LIN {X 0,Y 270.162,Z 852.684,A -85,B 0,C 180,E1 7695.271,E2 7695.271} C_VEL
LIN {X 0,Y 259.155,Z 871.54,A -85,B 0,C 180,E1 7693.362,E2 7693.362} C_VEL
LIN {X 0,Y 247.271,Z 889.429,A -85,B 0,C 180,E1 7691.066,E2 7691.066} C_VEL
LIN {X 0,Y 235.05,Z 906.14,A -85,B 0,C 180,E1 7688.382,E2 7688.382} C_VEL
LIN {X 0,Y 222.958,Z 921.018,A -85,B 0,C 180,E1 7685.334,E2 7685.334} C_VEL
LIN {X 0,Y 210.174,Z 935.544,A -85,B 0,C 180,E1 7681.543,E2 7681.543} C_VEL
LIN {X 0,Y 198.279,Z 948.046,A -85,B 0,C 180,E1 7677.304,E2 7677.304} C_VEL
LIN {X 0,Y 186.376,Z 959.885,A -85,B 0,C 180,E1 7672.046,E2 7672.046} C_VEL
LIN {X 0,Y 176.439,Z 969.458,A -85,B 0,C 180,E1 7666.449,E2 7666.449} C_VEL
LIN {X 0,Y 167.3,Z 978.146,A -85,B 0,C 180,E1 7659.622,E2 7659.622} C_VEL
LIN {X 0,Y 160.302,Z 985.227,A -85,B 0,C 180,E1 7652.134,E2 7652.134} C_VEL
LIN {X 0,Y 155.686,Z 990.327,A -85,B 0,C 180,E1 7644.461,E2 7644.461} C_VEL
LIN {X 0,Y 153.174,Z 993.985,A -85,B 0,C 180,E1 7636.782,E2 7636.782} C_VEL
LIN {X 0,Y 152.199,Z 996.255,A -85,B 0,C 180,E1 7628.889,E2 7628.889} C_VEL
LIN {X 0,Y 152.061,Z 997.122,A -85,B 0,C 180,E1 7623.007,E2 7623.007} C_VEL
LIN {X 0,Y 152.146,Z 997.282,A -85,B 0,C 180,E1 7616.932,E2 7616.932} C_VEL
LIN {X 0,Y 152.676,Z 996.667,A -85,B 0,C 180,E1 7610.549,E2 7610.549} C_VEL
LIN {X 0,Y 154.828,Z 994.686,A -85,B 0,C 180,E1 7602.194,E2 7602.194} C_VEL
LIN {X 0,Y 159.181,Z 991.12,A -85,B 0,C 180,E1 7593.974,E2 7593.974} C_VEL
LIN {X 0,Y 166.545,Z 985.817,A -85,B 0,C 180,E1 7585.753,E2 7585.753} C_VEL
LIN {X 0,Y 176.186,Z 979.026,A -85,B 0,C 180,E1 7578.531,E2 7578.531} C_VEL
LIN {X 0,Y 188.917,Z 969.957,A -85,B 0,C 180,E1 7571.693,E2 7571.693} C_VEL
LIN {X 0,Y 203.113,Z 959.499,A -85,B 0,C 180,E1 7566.019,E2 7566.019} C_VEL
LIN {X 0,Y 218.195,Z 947.498,A -85,B 0,C 180,E1 7561.314,E2 7561.314} C_VEL
LIN {X 0,Y 234.781,Z 933.271,A -85,B 0,C 180,E1 7557.194,E2 7557.194} C_VEL
LIN {X 0,Y 250.793,Z 918.312,A -85,B 0,C 180,E1 7553.948,E2 7553.948} C_VEL
LIN {X 0,Y 266.015,Z 902.433,A -85,B 0,C 180,E1 7551.34,E2 7551.34} C_VEL
LIN {X 0,Y 281.745,Z 884.288,A -85,B 0,C 180,E1 7549.046,E2 7549.046} C_VEL
LIN {X 0,Y 295.555,Z 866.409,A -85,B 0,C 180,E1 7547.298,E2 7547.298} C_VEL
LIN {X 0,Y 302.047,Z 857.131,A -85,B 0,C 180,E1 7546.521,E2 7546.521} C_VEL
LIN {X 0,Y 290.09,Z 874.11,A -85,B 0,C 180,E1 7545.216,E2 7545.216} C_VEL
LIN {X 0,Y 285.508,Z 880.165,A -85,B 0,C 180,E1 7544.883,E2 7544.883} C_VEL
LIN {X 0,Y 272.533,Z 895.474,A -85,B 0,C 180,E1 7544.622,E2 7544.622} C_VEL
LIN {X 0,Y 267.468,Z 900.978,A -85,B 0,C 180,E1 7544.201,E2 7544.201} C_VEL
LIN {X 0,Y 252.345,Z 916.917,A -85,B 0,C 180,E1 7541.995,E2 7541.995} C_VEL
LIN {X 0,Y 235.551,Z 933.117,A -85,B 0,C 180,E1 7539.058,E2 7539.058} C_VEL
LIN {X 0,Y 220.329,Z 946.567,A -85,B 0,C 180,E1 7535.817,E2 7535.817} C_VEL
LIN {X 0,Y 203.797,Z 960.142,A -85,B 0,C 180,E1 7531.44,E2 7531.44} C_VEL
LIN {X 0,Y 189.339,Z 971.334,A -85,B 0,C 180,E1 7526.563,E2 7526.563} C_VEL
LIN {X 0,Y 175.331,Z 981.675,A -85,B 0,C 180,E1 7520.354,E2 7520.354} C_VEL
LIN {X 0,Y 163.608,Z 990.335,A -85,B 0,C 180,E1 7513.206,E2 7513.206} C_VEL
LIN {X 0,Y 154.524,Z 997.124,A -85,B 0,C 180,E1 7505.173,E2 7505.173} C_VEL
LIN {X 0,Y 148.144,Z 1002.572,A -85,B 0,C 180,E1 7496.033,E2 7496.033} C_VEL
LIN {X 0,Y 145.093,Z 1005.814,A -85,B 0,C 180,E1 7487.662,E2 7487.662} C_VEL
LIN {X 0,Y 144.092,Z 1007.682,A -85,B 0,C 180,E1 7479.831,E2 7479.831} C_VEL
LIN {X 0,Y 144.042,Z 1008.346,A -85,B 0,C 180,E1 7472.797,E2 7472.797} C_VEL
LIN {X 0,Y 144.047,Z 1008.068,A -85,B 0,C 180,E1 7466.829,E2 7466.829} C_VEL
LIN {X 0,Y 144.115,Z 1006.784,A -85,B 0,C 180,E1 7460.024,E2 7460.024} C_VEL
LIN {X 0,Y 145.002,Z 1004.362,A -85,B 0,C 180,E1 7452.765,E2 7452.765} C_VEL
LIN {X 0,Y 147.505,Z 1000.647,A -85,B 0,C 180,E1 7445.163,E2 7445.163} C_VEL
LIN {X 0,Y 152.755,Z 994.682,A -85,B 0,C 180,E1 7436.66,E2 7436.66} C_VEL
LIN {X 0,Y 159.808,Z 987.715,A -85,B 0,C 180,E1 7429.423,E2 7429.423} C_VEL
LIN {X 0,Y 169.417,Z 978.623,A -85,B 0,C 180,E1 7422.48,E2 7422.48} C_VEL
LIN {X 0,Y 180.465,Z 968.26,A -85,B 0,C 180,E1 7416.566,E2 7416.566} C_VEL
LIN {X 0,Y 192.416,Z 956.466,A -85,B 0,C 180,E1 7411.569,E2 7411.569} C_VEL
LIN {X 0,Y 205.608,Z 942.836,A -85,B 0,C 180,E1 7407.16,E2 7407.16} C_VEL
LIN {X 0,Y 218.285,Z 928.559,A -85,B 0,C 180,E1 7403.662,E2 7403.662} C_VEL
LIN {X 0,Y 231.669,Z 912.241,A -85,B 0,C 180,E1 7400.548,E2 7400.548} C_VEL
LIN {X 0,Y 243.409,Z 896.383,A -85,B 0,C 180,E1 7398.19,E2 7398.19} C_VEL
LIN {X 0,Y 256.695,Z 876.382,A -85,B 0,C 180,E1 7395.859,E2 7395.859} C_VEL
LIN {X 0,Y 268.011,Z 857.211,A -85,B 0,C 180,E1 7394.113,E2 7394.113} C_VEL
LIN {X 0,Y 278.538,Z 836.599,A -85,B 0,C 180,E1 7392.648,E2 7392.648} C_VEL
LIN {X 0,Y 288.142,Z 814.942,A -85,B 0,C 180,E1 7391.439,E2 7391.439} C_VEL
LIN {X 0,Y 295.909,Z 794.1,A -85,B 0,C 180,E1 7390.539,E2 7390.539} C_VEL
LIN {X 0,Y 303.26,Z 770.05,A -85,B 0,C 180,E1 7389.753,E2 7389.753} C_VEL
LIN {X 0,Y 308.805,Z 746.808,A -85,B 0,C 180,E1 7389.177,E2 7389.177} C_VEL
LIN {X 0,Y 312.638,Z 723.003,A -85,B 0,C 180,E1 7388.694,E2 7388.694} C_VEL
LIN {X 0,Y 326.224,Z 603.459,A -85,B 0,C 180,E1 7386.559,E2 7386.559} C_VEL
LIN {X 0,Y 322.526,Z 597.162,A -85,B 0,C 180,E1 7383.198,E2 7383.198} C_VEL
LIN {X 0,Y 320.23,Z 593.384,A -85,B 0,C 180,E1 7380.715,E2 7380.715} C_VEL
LIN {X 0,Y 317.941,Z 589.485,A -85,B 0,C 180,E1 7377.656,E2 7377.656} C_VEL
LIN {X 0,Y 315.609,Z 585.291,A -85,B 0,C 180,E1 7373.268,E2 7373.268} C_VEL
LIN {X 0,Y 313.967,Z 583.652,A -85,B 0,C 180,E1 7367.119,E2 7367.119} C_VEL
LIN {X 0,Y 314.171,Z 583.904,A -85,B 0,C 180,E1 7362.592,E2 7362.592} C_VEL
LIN {X 0,Y 315.683,Z 585.371,A -85,B 0,C 180,E1 7357.857,E2 7357.857} C_VEL
LIN {X 0,Y 318.646,Z 590.582,A -85,B 0,C 180,E1 7352.608,E2 7352.608} C_VEL
LIN {X 0,Y 321.436,Z 595.282,A -85,B 0,C 180,E1 7349.222,E2 7349.222} C_VEL
LIN {X 0,Y 324.307,Z 600.175,A -85,B 0,C 180,E1 7346.387,E2 7346.387} C_VEL
LIN {X 0,Y 325.927,Z 603.009,A -85,B 0,C 180,E1 7344.966,E2 7344.966} C_VEL
LIN {X 0,Y 312.184,Z 722.288,A -85,B 0,C 180,E1 7342.851,E2 7342.851} C_VEL
LIN {X 0,Y 307.763,Z 746.045,A -85,B 0,C 180,E1 7342.322,E2 7342.322} C_VEL
LIN {X 0,Y 302.328,Z 768.096,A -85,B 0,C 180,E1 7341.675,E2 7341.675} C_VEL
LIN {X 0,Y 295.325,Z 790.127,A -85,B 0,C 180,E1 7340.821,E2 7340.821} C_VEL
LIN {X 0,Y 286.506,Z 813.129,A -85,B 0,C 180,E1 7339.676,E2 7339.676} C_VEL
LIN {X 0,Y 277.365,Z 833.259,A -85,B 0,C 180,E1 7338.406,E2 7338.406} C_VEL
LIN {X 0,Y 266.708,Z 853.445,A -85,B 0,C 180,E1 7336.804,E2 7336.804} C_VEL
LIN {X 0,Y 255.463,Z 872.302,A -85,B 0,C 180,E1 7334.936,E2 7334.936} C_VEL
LIN {X 0,Y 243.293,Z 890.156,A -85,B 0,C 180,E1 7332.683,E2 7332.683} C_VEL
LIN {X 0,Y 230.369,Z 907.254,A -85,B 0,C 180,E1 7329.956,E2 7329.956} C_VEL
LIN {X 0,Y 217.938,Z 922.067,A -85,B 0,C 180,E1 7326.93,E2 7326.93} C_VEL
LIN {X 0,Y 204.075,Z 937.188,A -85,B 0,C 180,E1 7322.934,E2 7322.934} C_VEL
LIN {X 0,Y 191.817,Z 949.595,A -85,B 0,C 180,E1 7318.645,E2 7318.645} C_VEL
LIN {X 0,Y 179.49,Z 961.211,A -85,B 0,C 180,E1 7313.286,E2 7313.286} C_VEL
LIN {X 0,Y 168.711,Z 971.103,A -85,B 0,C 180,E1 7307.225,E2 7307.225} C_VEL
LIN {X 0,Y 159.593,Z 979.245,A -85,B 0,C 180,E1 7300.379,E2 7300.379} C_VEL
LIN {X 0,Y 152.097,Z 986.35,A -85,B 0,C 180,E1 7292.224,E2 7292.224} C_VEL
LIN {X 0,Y 147.629,Z 991.075,A -85,B 0,C 180,E1 7284.547,E2 7284.547} C_VEL
LIN {X 0,Y 145.011,Z 994.73,A -85,B 0,C 180,E1 7276.023,E2 7276.023} C_VEL
LIN {X 0,Y 144.201,Z 996.581,A -85,B 0,C 180,E1 7268.853,E2 7268.853} C_VEL
LIN {X 0,Y 144.069,Z 997.435,A -85,B 0,C 180,E1 7262.669,E2 7262.669} C_VEL
LIN {X 0,Y 144.157,Z 997.607,A -85,B 0,C 180,E1 7256.762,E2 7256.762} C_VEL
LIN {X 0,Y 144.755,Z 997.043,A -85,B 0,C 180,E1 7250.017,E2 7250.017} C_VEL
LIN {X 0,Y 147.012,Z 995.246,A -85,B 0,C 180,E1 7241.556,E2 7241.556} C_VEL
LIN {X 0,Y 151.941,Z 991.659,A -85,B 0,C 180,E1 7232.597,E2 7232.597} C_VEL
LIN {X 0,Y 159.924,Z 986.487,A -85,B 0,C 180,E1 7224.083,E2 7224.083} C_VEL
LIN {X 0,Y 170.496,Z 979.611,A -85,B 0,C 180,E1 7216.529,E2 7216.529} C_VEL
LIN {X 0,Y 184.493,Z 970.332,A -85,B 0,C 180,E1 7209.435,E2 7209.435} C_VEL
LIN {X 0,Y 199.438,Z 959.955,A -85,B 0,C 180,E1 7203.823,E2 7203.823} C_VEL
LIN {X 0,Y 215.272,Z 947.978,A -85,B 0,C 180,E1 7199.203,E2 7199.203} C_VEL
LIN {X 0,Y 232.015,Z 934.265,A -85,B 0,C 180,E1 7195.304,E2 7195.304} C_VEL
LIN {X 0,Y 248.645,Z 919.344,A -85,B 0,C 180,E1 7192.143,E2 7192.143} C_VEL
LIN {X 0,Y 264.823,Z 903.077,A -85,B 0,C 180,E1 7189.56,E2 7189.56} C_VEL
LIN {X 0,Y 280.736,Z 885.326,A -85,B 0,C 180,E1 7187.405,E2 7187.405} C_VEL
LIN {X 0,Y 287.244,Z 877.461,A -85,B 0,C 180,E1 7186.594,E2 7186.594} C_VEL
LIN {X 0,Y 273.077,Z 894.577,A -85,B 0,C 180,E1 7184.933,E2 7184.933} C_VEL
LIN {X 0,Y 267.468,Z 900.978,A -85,B 0,C 180,E1 7184.201,E2 7184.201} C_VEL
LIN {X 0,Y 262.279,Z 906.461,A -85,B 0,C 180,E1 7183.741,E2 7183.741} C_VEL
LIN {X 0,Y 247.934,Z 920.355,A -85,B 0,C 180,E1 7183.165,E2 7183.165} C_VEL
LIN {X 0,Y 242.565,Z 925.2,A -85,B 0,C 180,E1 7182.583,E2 7182.583} C_VEL
LIN {X 0,Y 225.228,Z 940.622,A -85,B 0,C 180,E1 7179.471,E2 7179.471} C_VEL
LIN {X 0,Y 208.402,Z 954.183,A -85,B 0,C 180,E1 7175.739,E2 7175.739} C_VEL
LIN {X 0,Y 190.481,Z 967.605,A -85,B 0,C 180,E1 7170.631,E2 7170.631} C_VEL
LIN {X 0,Y 174.945,Z 978.613,A -85,B 0,C 180,E1 7164.745,E2 7164.745} C_VEL
LIN {X 0,Y 161.697,Z 987.525,A -85,B 0,C 180,E1 7157.918,E2 7157.918} C_VEL
LIN {X 0,Y 150.354,Z 995.281,A -85,B 0,C 180,E1 7149.522,E2 7149.522} C_VEL
LIN {X 0,Y 142.712,Z 1000.798,A -85,B 0,C 180,E1 7140.773,E2 7140.773} C_VEL
LIN {X 0,Y 137.876,Z 1004.997,A -85,B 0,C 180,E1 7130.697,E2 7130.697} C_VEL
LIN {X 0,Y 136.278,Z 1007.009,A -85,B 0,C 180,E1 7122.636,E2 7122.636} C_VEL
LIN {X 0,Y 136.032,Z 1007.885,A -85,B 0,C 180,E1 7115.496,E2 7115.496} C_VEL
LIN {X 0,Y 136.079,Z 1007.881,A -85,B 0,C 180,E1 7109.171,E2 7109.171} C_VEL
LIN {X 0,Y 136.04,Z 1007.111,A -85,B 0,C 180,E1 7102.833,E2 7102.833} C_VEL
LIN {X 0,Y 136.628,Z 1005.093,A -85,B 0,C 180,E1 7094.739,E2 7094.739} C_VEL
LIN {X 0,Y 139.031,Z 1001.332,A -85,B 0,C 180,E1 7085.966,E2 7085.966} C_VEL
LIN {X 0,Y 143.696,Z 996.28,A -85,B 0,C 180,E1 7077.619,E2 7077.619} C_VEL
LIN {X 0,Y 150.992,Z 989.347,A -85,B 0,C 180,E1 7069.555,E2 7069.555} C_VEL
LIN {X 0,Y 160.748,Z 980.735,A -85,B 0,C 180,E1 7062.201,E2 7062.201} C_VEL
LIN {X 0,Y 172.157,Z 970.459,A -85,B 0,C 180,E1 7055.914,E2 7055.914} C_VEL
LIN {X 0,Y 185.372,Z 958.223,A -85,B 0,C 180,E1 7050.367,E2 7050.367} C_VEL
LIN {X 0,Y 198.608,Z 945.144,A -85,B 0,C 180,E1 7045.974,E2 7045.974} C_VEL
LIN {X 0,Y 212.657,Z 930.054,A -85,B 0,C 180,E1 7042.171,E2 7042.171} C_VEL
LIN {X 0,Y 226.361,Z 914.035,A -85,B 0,C 180,E1 7039.076,E2 7039.076} C_VEL
LIN {X 0,Y 239.354,Z 896.996,A -85,B 0,C 180,E1 7036.559,E2 7036.559} C_VEL
LIN {X 0,Y 252.328,Z 878.125,A -85,B 0,C 180,E1 7034.377,E2 7034.377} C_VEL
LIN {X 0,Y 263.801,Z 859.218,A -85,B 0,C 180,E1 7032.674,E2 7032.674} C_VEL
LIN {X 0,Y 274.861,Z 838.315,A -85,B 0,C 180,E1 7031.2,E2 7031.2} C_VEL
LIN {X 0,Y 284.294,Z 817.819,A -85,B 0,C 180,E1 7030.065,E2 7030.065} C_VEL
LIN {X 0,Y 292.631,Z 796.13,A -85,B 0,C 180,E1 7029.138,E2 7029.138} C_VEL
LIN {X 0,Y 299.852,Z 773.653,A -85,B 0,C 180,E1 7028.402,E2 7028.402} C_VEL
LIN {X 0,Y 305.465,Z 751.2,A -85,B 0,C 180,E1 7027.85,E2 7027.85} C_VEL
LIN {X 0,Y 309.952,Z 726.087,A -85,B 0,C 180,E1 7027.337,E2 7027.337} C_VEL
LIN {X 0,Y 323.595,Z 609.157,A -85,B 0,C 180,E1 7025.274,E2 7025.274} C_VEL
LIN {X 0,Y 320.64,Z 604.095,A -85,B 0,C 180,E1 7022.412,E2 7022.412} C_VEL
LIN {X 0,Y 318.812,Z 601.022,A -85,B 0,C 180,E1 7020.359,E2 7020.359} C_VEL
LIN {X 0,Y 316.708,Z 597.319,A -85,B 0,C 180,E1 7017.466,E2 7017.466} C_VEL
LIN {X 0,Y 314.42,Z 593.131,A -85,B 0,C 180,E1 7013.059,E2 7013.059} C_VEL
LIN {X 0,Y 312.859,Z 591.556,A -85,B 0,C 180,E1 7006.884,E2 7006.884} C_VEL
LIN {X 0,Y 313.119,Z 591.891,A -85,B 0,C 180,E1 7002.34,E2 7002.34} C_VEL
LIN {X 0,Y 314.525,Z 593.322,A -85,B 0,C 180,E1 6997.968,E2 6997.968} C_VEL
LIN {X 0,Y 317.37,Z 598.423,A -85,B 0,C 180,E1 6992.817,E2 6992.817} C_VEL
LIN {X 0,Y 320.048,Z 603.022,A -85,B 0,C 180,E1 6989.501,E2 6989.501} C_VEL
LIN {X 0,Y 322.87,Z 607.937,A -85,B 0,C 180,E1 6986.654,E2 6986.654} C_VEL
LIN {X 0,Y 323.29,Z 608.915,A -85,B 0,C 180,E1 6986.237,E2 6986.237} C_VEL
LIN {X 0,Y 309.904,Z 722.563,A -85,B 0,C 180,E1 6984.262,E2 6984.262} C_VEL
LIN {X 0,Y 305.413,Z 746.343,A -85,B 0,C 180,E1 6983.751,E2 6983.751} C_VEL
LIN {X 0,Y 299.702,Z 769.038,A -85,B 0,C 180,E1 6983.103,E2 6983.103} C_VEL
LIN {X 0,Y 293.013,Z 789.796,A -85,B 0,C 180,E1 6982.328,E2 6982.328} C_VEL
LIN {X 0,Y 284.468,Z 811.998,A -85,B 0,C 180,E1 6981.275,E2 6981.275} C_VEL
LIN {X 0,Y 275.151,Z 832.32,A -85,B 0,C 180,E1 6980.05,E2 6980.05} C_VEL
LIN {X 0,Y 263.86,Z 853.451,A -85,B 0,C 180,E1 6978.439,E2 6978.439} C_VEL
LIN {X 0,Y 251.96,Z 872.97,A -85,B 0,C 180,E1 6976.557,E2 6976.557} C_VEL
LIN {X 0,Y 239.505,Z 890.788,A -85,B 0,C 180,E1 6974.355,E2 6974.355} C_VEL
LIN {X 0,Y 225.865,Z 908.325,A -85,B 0,C 180,E1 6971.595,E2 6971.595} C_VEL
LIN {X 0,Y 213.094,Z 923.108,A -85,B 0,C 180,E1 6968.6,E2 6968.6} C_VEL
LIN {X 0,Y 199.488,Z 937.426,A -85,B 0,C 180,E1 6964.834,E2 6964.834} C_VEL
LIN {X 0,Y 186.739,Z 949.846,A -85,B 0,C 180,E1 6960.562,E2 6960.562} C_VEL
LIN {X 0,Y 173.848,Z 961.488,A -85,B 0,C 180,E1 6955.176,E2 6955.176} C_VEL
LIN {X 0,Y 162.484,Z 971.404,A -85,B 0,C 180,E1 6949.023,E2 6949.023} C_VEL
LIN {X 0,Y 152.887,Z 979.481,A -85,B 0,C 180,E1 6942.068,E2 6942.068} C_VEL
LIN {X 0,Y 145.085,Z 986.383,A -85,B 0,C 180,E1 6933.94,E2 6933.94} C_VEL
LIN {X 0,Y 140.126,Z 991.169,A -85,B 0,C 180,E1 6925.896,E2 6925.896} C_VEL
LIN {X 0,Y 137.17,Z 994.917,A -85,B 0,C 180,E1 6916.928,E2 6916.928} C_VEL
LIN {X 0,Y 136.202,Z 996.904,A -85,B 0,C 180,E1 6908.802,E2 6908.802} C_VEL
LIN {X 0,Y 136.075,Z 997.737,A -85,B 0,C 180,E1 6902.411,E2 6902.411} C_VEL
LIN {X 0,Y 136.189,Z 997.917,A -85,B 0,C 180,E1 6896.062,E2 6896.062} C_VEL
LIN {X 0,Y 136.958,Z 997.335,A -85,B 0,C 180,E1 6888.762,E2 6888.762} C_VEL
LIN {X 0,Y 139.749,Z 995.455,A -85,B 0,C 180,E1 6879.553,E2 6879.553} C_VEL
LIN {X 0,Y 145.197,Z 991.97,A -85,B 0,C 180,E1 6870.577,E2 6870.577} C_VEL
LIN {X 0,Y 154.127,Z 986.734,A -85,B 0,C 180,E1 6861.703,E2 6861.703} C_VEL
LIN {X 0,Y 165.137,Z 980.154,A -85,B 0,C 180,E1 6854.326,E2 6854.326} C_VEL
LIN {X 0,Y 179.687,Z 971.191,A -85,B 0,C 180,E1 6847.354,E2 6847.354} C_VEL
LIN {X 0,Y 194.432,Z 961.539,A -85,B 0,C 180,E1 6842.064,E2 6842.064} C_VEL
LIN {X 0,Y 210.567,Z 950.06,A -85,B 0,C 180,E1 6837.552,E2 6837.552} C_VEL
LIN {X 0,Y 227.311,Z 937.188,A -85,B 0,C 180,E1 6833.819,E2 6833.819} C_VEL
LIN {X 0,Y 243.785,Z 923.052,A -85,B 0,C 180,E1 6830.797,E2 6830.797} C_VEL
LIN {X 0,Y 260.438,Z 907.351,A -85,B 0,C 180,E1 6828.253,E2 6828.253} C_VEL
LIN {X 0,Y 272.321,Z 894.975,A -85,B 0,C 180,E1 6826.668,E2 6826.668} C_VEL
LIN {X 0,Y 255.283,Z 912.982,A -85,B 0,C 180,E1 6824.489,E2 6824.489} C_VEL
LIN {X 0,Y 242.565,Z 925.2,A -85,B 0,C 180,E1 6822.583,E2 6822.583} C_VEL
LIN {X 0,Y 237.076,Z 930.151,A -85,B 0,C 180,E1 6821.949,E2 6821.949} C_VEL
LIN {X 0,Y 221.601,Z 942.319,A -85,B 0,C 180,E1 6820.953,E2 6820.953} C_VEL
LIN {X 0,Y 215.982,Z 946.624,A -85,B 0,C 180,E1 6820.166,E2 6820.166} C_VEL
LIN {X 0,Y 198.015,Z 960.01,A -85,B 0,C 180,E1 6816.072,E2 6816.072} C_VEL
LIN {X 0,Y 180.739,Z 972.007,A -85,B 0,C 180,E1 6810.95,E2 6810.95} C_VEL
LIN {X 0,Y 165.19,Z 981.995,A -85,B 0,C 180,E1 6804.813,E2 6804.813} C_VEL
LIN {X 0,Y 150.825,Z 990.968,A -85,B 0,C 180,E1 6796.835,E2 6796.835} C_VEL
LIN {X 0,Y 140.443,Z 997.516,A -85,B 0,C 180,E1 6788.285,E2 6788.285} C_VEL
LIN {X 0,Y 132.973,Z 1002.569,A -85,B 0,C 180,E1 6778.289,E2 6778.289} C_VEL
LIN {X 0,Y 129.324,Z 1005.632,A -85,B 0,C 180,E1 6768.962,E2 6768.962} C_VEL
LIN {X 0,Y 128.086,Z 1007.33,A -85,B 0,C 180,E1 6759.448,E2 6759.448} C_VEL
LIN {X 0,Y 128.07,Z 1007.674,A -85,B 0,C 180,E1 6752.173,E2 6752.173} C_VEL
LIN {X 0,Y 128.056,Z 1007.296,A -85,B 0,C 180,E1 6745.984,E2 6745.984} C_VEL
LIN {X 0,Y 128.18,Z 1006.002,A -85,B 0,C 180,E1 6738.769,E2 6738.769} C_VEL
LIN {X 0,Y 129.433,Z 1003.5,A -85,B 0,C 180,E1 6730.614,E2 6730.614} C_VEL
LIN {X 0,Y 133.113,Z 999.24,A -85,B 0,C 180,E1 6721.283,E2 6721.283} C_VEL
LIN {X 0,Y 139.451,Z 993.223,A -85,B 0,C 180,E1 6712.468,E2 6712.468} C_VEL
LIN {X 0,Y 148.404,Z 985.668,A -85,B 0,C 180,E1 6704.444,E2 6704.444} C_VEL
LIN {X 0,Y 159.468,Z 976.363,A -85,B 0,C 180,E1 6697.457,E2 6697.457} C_VEL
LIN {X 0,Y 172.921,Z 964.773,A -85,B 0,C 180,E1 6691.179,E2 6691.179} C_VEL
LIN {X 0,Y 186.317,Z 952.571,A -85,B 0,C 180,E1 6686.363,E2 6686.363} C_VEL
LIN {X 0,Y 200.413,Z 938.594,A -85,B 0,C 180,E1 6682.281,E2 6682.281} C_VEL
LIN {X 0,Y 214.524,Z 923.448,A -85,B 0,C 180,E1 6678.921,E2 6678.921} C_VEL
LIN {X 0,Y 227.995,Z 907.301,A -85,B 0,C 180,E1 6676.211,E2 6676.211} C_VEL
LIN {X 0,Y 241.917,Z 888.754,A -85,B 0,C 180,E1 6673.806,E2 6673.806} C_VEL
LIN {X 0,Y 253.964,Z 870.686,A -85,B 0,C 180,E1 6671.988,E2 6671.988} C_VEL
LIN {X 0,Y 265.75,Z 850.531,A -85,B 0,C 180,E1 6670.404,E2 6670.404} C_VEL
LIN {X 0,Y 276.413,Z 829.703,A -85,B 0,C 180,E1 6669.118,E2 6669.118} C_VEL
LIN {X 0,Y 285.761,Z 807.984,A -85,B 0,C 180,E1 6668.088,E2 6668.088} C_VEL
LIN {X 0,Y 294.382,Z 783.947,A -85,B 0,C 180,E1 6667.219,E2 6667.219} C_VEL
LIN {X 0,Y 301.07,Z 760.838,A -85,B 0,C 180,E1 6666.605,E2 6666.605} C_VEL
LIN {X 0,Y 306.053,Z 737.258,A -85,B 0,C 180,E1 6666.115,E2 6666.115} C_VEL
LIN {X 0,Y 310.281,Z 706.846,A -85,B 0,C 180,E1 6665.563,E2 6665.563} C_VEL
LIN {X 0,Y 321.009,Z 614.994,A -85,B 0,C 180,E1 6663.973,E2 6663.973} C_VEL
LIN {X 0,Y 317.843,Z 609.291,A -85,B 0,C 180,E1 6660.54,E2 6660.54} C_VEL
LIN {X 0,Y 315.332,Z 604.972,A -85,B 0,C 180,E1 6657.043,E2 6657.043} C_VEL
LIN {X 0,Y 313.083,Z 600.816,A -85,B 0,C 180,E1 6652.476,E2 6652.476} C_VEL
LIN {X 0,Y 311.752,Z 599.412,A -85,B 0,C 180,E1 6646.081,E2 6646.081} C_VEL
LIN {X 0,Y 312.294,Z 600.153,A -85,B 0,C 180,E1 6641.133,E2 6641.133} C_VEL
LIN {X 0,Y 313.324,Z 601.133,A -85,B 0,C 180,E1 6638.2,E2 6638.2} C_VEL
LIN {X 0,Y 316.049,Z 606.16,A -85,B 0,C 180,E1 6633.102,E2 6633.102} C_VEL
LIN {X 0,Y 318.587,Z 610.634,A -85,B 0,C 180,E1 6629.857,E2 6629.857} C_VEL
LIN {X 0,Y 320.773,Z 614.625,A -85,B 0,C 180,E1 6627.529,E2 6627.529} C_VEL
LIN {X 0,Y 307.787,Z 723,A -85,B 0,C 180,E1 6625.691,E2 6625.691} C_VEL
LIN {X 0,Y 303.253,Z 746.596,A -85,B 0,C 180,E1 6625.201,E2 6625.201} C_VEL
LIN {X 0,Y 297.48,Z 769.205,A -85,B 0,C 180,E1 6624.58,E2 6624.58} C_VEL
LIN {X 0,Y 290.47,Z 790.589,A -85,B 0,C 180,E1 6623.81,E2 6623.81} C_VEL
LIN {X 0,Y 281.782,Z 812.684,A -85,B 0,C 180,E1 6622.794,E2 6622.794} C_VEL
LIN {X 0,Y 272.303,Z 832.967,A -85,B 0,C 180,E1 6621.61,E2 6621.61} C_VEL
LIN {X 0,Y 261.225,Z 853.354,A -85,B 0,C 180,E1 6620.11,E2 6620.11} C_VEL
LIN {X 0,Y 249.487,Z 872.331,A -85,B 0,C 180,E1 6618.355,E2 6618.355} C_VEL
LIN {X 0,Y 236.737,Z 890.324,A -85,B 0,C 180,E1 6616.225,E2 6616.225} C_VEL
LIN {X 0,Y 223.914,Z 906.63,A -85,B 0,C 180,E1 6613.786,E2 6613.786} C_VEL
LIN {X 0,Y 209.945,Z 922.42,A -85,B 0,C 180,E1 6610.714,E2 6610.714} C_VEL
LIN {X 0,Y 195.127,Z 937.619,A -85,B 0,C 180,E1 6606.823,E2 6606.823} C_VEL
LIN {X 0,Y 181.88,Z 950.078,A -85,B 0,C 180,E1 6602.585,E2 6602.585} C_VEL
LIN {X 0,Y 169.018,Z 961.239,A -85,B 0,C 180,E1 6597.466,E2 6597.466} C_VEL
LIN {X 0,Y 156.957,Z 971.25,A -85,B 0,C 180,E1 6591.278,E2 6591.278} C_VEL
LIN {X 0,Y 146.231,Z 979.762,A -85,B 0,C 180,E1 6583.833,E2 6583.833} C_VEL
LIN {X 0,Y 137.858,Z 986.68,A -85,B 0,C 180,E1 6575.397,E2 6575.397} C_VEL
LIN {X 0,Y 132.492,Z 991.472,A -85,B 0,C 180,E1 6566.959,E2 6566.959} C_VEL
LIN {X 0,Y 129.261,Z 995.22,A -85,B 0,C 180,E1 6557.478,E2 6557.478} C_VEL
LIN {X 0,Y 128.214,Z 997.191,A -85,B 0,C 180,E1 6548.964,E2 6548.964} C_VEL
LIN {X 0,Y 128.087,Z 998.055,A -85,B 0,C 180,E1 6541.899,E2 6541.899} C_VEL
LIN {X 0,Y 128.23,Z 998.229,A -85,B 0,C 180,E1 6535.29,E2 6535.29} C_VEL
LIN {X 0,Y 129.226,Z 997.629,A -85,B 0,C 180,E1 6527.313,E2 6527.313} C_VEL
LIN {X 0,Y 132.529,Z 995.727,A -85,B 0,C 180,E1 6517.593,E2 6517.593} C_VEL
LIN {X 0,Y 139.093,Z 992.054,A -85,B 0,C 180,E1 6507.827,E2 6507.827} C_VEL
LIN {X 0,Y 149.115,Z 986.721,A -85,B 0,C 180,E1 6498.777,E2 6498.777} C_VEL
LIN {X 0,Y 161.173,Z 980.112,A -85,B 0,C 180,E1 6491.384,E2 6491.384} C_VEL
LIN {X 0,Y 176.735,Z 971.107,A -85,B 0,C 180,E1 6484.544,E2 6484.544} C_VEL
LIN {X 0,Y 193.013,Z 961.035,A -85,B 0,C 180,E1 6479.23,E2 6479.23} C_VEL
LIN {X 0,Y 209.804,Z 949.517,A -85,B 0,C 180,E1 6474.96,E2 6474.96} C_VEL
LIN {X 0,Y 227.351,Z 936.411,A -85,B 0,C 180,E1 6471.401,E2 6471.401} C_VEL
LIN {X 0,Y 243.869,Z 922.688,A -85,B 0,C 180,E1 6468.651,E2 6468.651} C_VEL
LIN {X 0,Y 257.25,Z 910.597,A -85,B 0,C 180,E1 6466.72,E2 6466.72} C_VEL
LIN {X 0,Y 240.773,Z 925.935,A -85,B 0,C 180,E1 6464.475,E2 6464.475} C_VEL
LIN {X 0,Y 221.721,Z 942.067,A -85,B 0,C 180,E1 6461.28,E2 6461.28} C_VEL
LIN {X 0,Y 215.982,Z 946.624,A -85,B 0,C 180,E1 6460.166,E2 6460.166} C_VEL
LIN {X 0,Y 210.309,Z 950.884,A -85,B 0,C 180,E1 6459.312,E2 6459.312} C_VEL
LIN {X 0,Y 194.107,Z 961.41,A -85,B 0,C 180,E1 6457.719,E2 6457.719} C_VEL
LIN {X 0,Y 188.3,Z 965.007,A -85,B 0,C 180,E1 6456.622,E2 6456.622} C_VEL
LIN {X 0,Y 171.693,Z 975.494,A -85,B 0,C 180,E1 6451.581,E2 6451.581} C_VEL
LIN {X 0,Y 154.706,Z 985.598,A -85,B 0,C 180,E1 6444.538,E2 6444.538} C_VEL
LIN {X 0,Y 141.511,Z 993.168,A -85,B 0,C 180,E1 6436.714,E2 6436.714} C_VEL
LIN {X 0,Y 130.835,Z 999.269,A -85,B 0,C 180,E1 6427.152,E2 6427.152} C_VEL
LIN {X 0,Y 124.037,Z 1003.616,A -85,B 0,C 180,E1 6416.849,E2 6416.849} C_VEL
LIN {X 0,Y 120.715,Z 1006.212,A -85,B 0,C 180,E1 6406.101,E2 6406.101} C_VEL
LIN {X 0,Y 120.033,Z 1007.218,A -85,B 0,C 180,E1 6397.597,E2 6397.597} C_VEL
LIN {X 0,Y 120.09,Z 1007.309,A -85,B 0,C 180,E1 6390.969,E2 6390.969} C_VEL
LIN {X 0,Y 120.059,Z 1006.802,A -85,B 0,C 180,E1 6384.759,E2 6384.759} C_VEL
LIN {X 0,Y 120.273,Z 1005.482,A -85,B 0,C 180,E1 6377.533,E2 6377.533} C_VEL
LIN {X 0,Y 121.861,Z 1002.883,A -85,B 0,C 180,E1 6368.854,E2 6368.854} C_VEL
LIN {X 0,Y 126.43,Z 998.163,A -85,B 0,C 180,E1 6358.554,E2 6358.554} C_VEL
LIN {X 0,Y 133.319,Z 992.313,A -85,B 0,C 180,E1 6349.855,E2 6349.855} C_VEL
LIN {X 0,Y 144.231,Z 983.677,A -85,B 0,C 180,E1 6340.941,E2 6340.941} C_VEL
LIN {X 0,Y 156.588,Z 973.948,A -85,B 0,C 180,E1 6333.916,E2 6333.916} C_VEL
LIN {X 0,Y 170.118,Z 962.644,A -85,B 0,C 180,E1 6328.188,E2 6328.188} C_VEL
LIN {X 0,Y 185.021,Z 949.395,A -85,B 0,C 180,E1 6323.295,E2 6323.295} C_VEL
LIN {X 0,Y 198.569,Z 936.219,A -85,B 0,C 180,E1 6319.71,E2 6319.71} C_VEL
LIN {X 0,Y 213.638,Z 920.119,A -85,B 0,C 180,E1 6316.413,E2 6316.413} C_VEL
LIN {X 0,Y 227.547,Z 903.669,A -85,B 0,C 180,E1 6313.852,E2 6313.852} C_VEL
LIN {X 0,Y 240.947,Z 885.738,A -85,B 0,C 180,E1 6311.717,E2 6311.717} C_VEL
LIN {X 0,Y 253.731,Z 866.567,A -85,B 0,C 180,E1 6309.938,E2 6309.938} C_VEL
LIN {X 0,Y 264.868,Z 847.356,A -85,B 0,C 180,E1 6308.554,E2 6308.554} C_VEL
LIN {X 0,Y 275.681,Z 825.893,A -85,B 0,C 180,E1 6307.343,E2 6307.343} C_VEL
LIN {X 0,Y 284.291,Z 805.886,A -85,B 0,C 180,E1 6306.461,E2 6306.461} C_VEL
LIN {X 0,Y 292.458,Z 783.064,A -85,B 0,C 180,E1 6305.689,E2 6305.689} C_VEL
LIN {X 0,Y 299.198,Z 759.867,A -85,B 0,C 180,E1 6305.109,E2 6305.109} C_VEL
LIN {X 0,Y 304.164,Z 736.516,A -85,B 0,C 180,E1 6304.645,E2 6304.645} C_VEL
LIN {X 0,Y 308.524,Z 705.365,A -85,B 0,C 180,E1 6304.097,E2 6304.097} C_VEL
LIN {X 0,Y 318.642,Z 620.838,A -85,B 0,C 180,E1 6302.697,E2 6302.697} C_VEL
LIN {X 0,Y 316.07,Z 616.401,A -85,B 0,C 180,E1 6299.727,E2 6299.727} C_VEL
LIN {X 0,Y 314.125,Z 612.842,A -85,B 0,C 180,E1 6296.897,E2 6296.897} C_VEL
LIN {X 0,Y 311.905,Z 608.688,A -85,B 0,C 180,E1 6292.262,E2 6292.262} C_VEL
LIN {X 0,Y 310.661,Z 607.335,A -85,B 0,C 180,E1 6286.031,E2 6286.031} C_VEL
LIN {X 0,Y 311.22,Z 608.101,A -85,B 0,C 180,E1 6281.065,E2 6281.065} C_VEL
LIN {X 0,Y 312.145,Z 608.999,A -85,B 0,C 180,E1 6278.384,E2 6278.384} C_VEL
LIN {X 0,Y 314.734,Z 613.896,A -85,B 0,C 180,E1 6273.388,E2 6273.388} C_VEL
LIN {X 0,Y 317.207,Z 618.388,A -85,B 0,C 180,E1 6270.13,E2 6270.13} C_VEL
LIN {X 0,Y 318.348,Z 620.654,A -85,B 0,C 180,E1 6268.835,E2 6268.835} C_VEL
LIN {X 0,Y 305.794,Z 723.263,A -85,B 0,C 180,E1 6267.138,E2 6267.138} C_VEL
LIN {X 0,Y 301.167,Z 746.997,A -85,B 0,C 180,E1 6266.663,E2 6266.663} C_VEL
LIN {X 0,Y 295.228,Z 769.866,A -85,B 0,C 180,E1 6266.059,E2 6266.059} C_VEL
LIN {X 0,Y 288.116,Z 791.241,A -85,B 0,C 180,E1 6265.319,E2 6265.319} C_VEL
LIN {X 0,Y 278.854,Z 814.273,A -85,B 0,C 180,E1 6264.291,E2 6264.291} C_VEL
LIN {X 0,Y 269.226,Z 834.467,A -85,B 0,C 180,E1 6263.148,E2 6263.148} C_VEL
LIN {X 0,Y 257.953,Z 854.658,A -85,B 0,C 180,E1 6261.699,E2 6261.699} C_VEL
LIN {X 0,Y 245.993,Z 873.522,A -85,B 0,C 180,E1 6259.998,E2 6259.998} C_VEL
LIN {X 0,Y 232.976,Z 891.392,A -85,B 0,C 180,E1 6257.928,E2 6257.928} C_VEL
LIN {X 0,Y 218.239,Z 909.425,A -85,B 0,C 180,E1 6255.232,E2 6255.232} C_VEL
LIN {X 0,Y 204.749,Z 924.206,A -85,B 0,C 180,E1 6252.355,E2 6252.355} C_VEL
LIN {X 0,Y 190.263,Z 938.485,A -85,B 0,C 180,E1 6248.695,E2 6248.695} C_VEL
LIN {X 0,Y 175.866,Z 951.514,A -85,B 0,C 180,E1 6244.24,E2 6244.24} C_VEL
LIN {X 0,Y 161.909,Z 962.992,A -85,B 0,C 180,E1 6238.782,E2 6238.782} C_VEL
LIN {X 0,Y 148.352,Z 973.546,A -85,B 0,C 180,E1 6231.745,E2 6231.745} C_VEL
LIN {X 0,Y 137.906,Z 981.457,A -85,B 0,C 180,E1 6224.257,E2 6224.257} C_VEL
LIN {X 0,Y 129.375,Z 987.993,A -85,B 0,C 180,E1 6215.308,E2 6215.308} C_VEL
LIN {X 0,Y 123.826,Z 992.822,A -85,B 0,C 180,E1 6205.819,E2 6205.819} C_VEL
LIN {X 0,Y 120.9,Z 996.114,A -85,B 0,C 180,E1 6195.62,E2 6195.62} C_VEL
LIN {X 0,Y 120.171,Z 997.644,A -85,B 0,C 180,E1 6187.997,E2 6187.997} C_VEL
LIN {X 0,Y 120.106,Z 998.394,A -85,B 0,C 180,E1 6180.943,E2 6180.943} C_VEL
LIN {X 0,Y 120.344,Z 998.525,A -85,B 0,C 180,E1 6173.702,E2 6173.702} C_VEL
LIN {X 0,Y 121.877,Z 997.789,A -85,B 0,C 180,E1 6164.443,E2 6164.443} C_VEL
LIN {X 0,Y 126.742,Z 995.331,A -85,B 0,C 180,E1 6153.235,E2 6153.235} C_VEL
LIN {X 0,Y 134.951,Z 991.438,A -85,B 0,C 180,E1 6143.232,E2 6143.232} C_VEL
LIN {X 0,Y 146.565,Z 985.713,A -85,B 0,C 180,E1 6134.33,E2 6134.33} C_VEL
LIN {X 0,Y 161.114,Z 978.311,A -85,B 0,C 180,E1 6126.739,E2 6126.739} C_VEL
LIN {X 0,Y 176.25,Z 969.939,A -85,B 0,C 180,E1 6120.976,E2 6120.976} C_VEL
LIN {X 0,Y 194.533,Z 958.929,A -85,B 0,C 180,E1 6115.739,E2 6115.739} C_VEL
LIN {X 0,Y 211.019,Z 948.024,A -85,B 0,C 180,E1 6112.052,E2 6112.052} C_VEL
LIN {X 0,Y 229.402,Z 934.497,A -85,B 0,C 180,E1 6108.744,E2 6108.744} C_VEL
LIN {X 0,Y 242.155,Z 924.237,A -85,B 0,C 180,E1 6106.78,E2 6106.78} C_VEL
LIN {X 0,Y 223.628,Z 939.653,A -85,B 0,C 180,E1 6104.025,E2 6104.025} C_VEL
LIN {X 0,Y 205.571,Z 953.103,A -85,B 0,C 180,E1 6100.681,E2 6100.681} C_VEL
LIN {X 0,Y 188.3,Z 965.007,A -85,B 0,C 180,E1 6096.622,E2 6096.622} C_VEL
LIN {X 0,Y 182.49,Z 968.519,A -85,B 0,C 180,E1 6095.434,E2 6095.434} C_VEL
LIN {X 0,Y 165.119,Z 977.698,A -85,B 0,C 180,E1 6092.769,E2 6092.769} C_VEL
LIN {X 0,Y 160.328,Z 980.138,A -85,B 0,C 180,E1 6091.417,E2 6091.417} C_VEL
LIN {X 0,Y 144.208,Z 988.923,A -85,B 0,C 180,E1 6084.232,E2 6084.232} C_VEL
LIN {X 0,Y 130.659,Z 995.879,A -85,B 0,C 180,E1 6075.388,E2 6075.388} C_VEL
LIN {X 0,Y 120.21,Z 1001.406,A -85,B 0,C 180,E1 6064.46,E2 6064.46} C_VEL
LIN {X 0,Y 114.77,Z 1004.594,A -85,B 0,C 180,E1 6054.186,E2 6054.186} C_VEL
LIN {X 0,Y 112.28,Z 1006.614,A -85,B 0,C 180,E1 6042.879,E2 6042.879} C_VEL
LIN {X 0,Y 112.051,Z 1007.073,A -85,B 0,C 180,E1 6034.109,E2 6034.109} C_VEL
LIN {X 0,Y 112.08,Z 1006.833,A -85,B 0,C 180,E1 6027.459,E2 6027.459} C_VEL
LIN {X 0,Y 112.157,Z 1005.66,A -85,B 0,C 180,E1 6019.226,E2 6019.226} C_VEL
LIN {X 0,Y 113.63,Z 1003.099,A -85,B 0,C 180,E1 6009.409,E2 6009.409} C_VEL
LIN {X 0,Y 117.669,Z 999.127,A -85,B 0,C 180,E1 5999.366,E2 5999.366} C_VEL
LIN {X 0,Y 125.293,Z 992.977,A -85,B 0,C 180,E1 5989.148,E2 5989.148} C_VEL
LIN {X 0,Y 135.631,Z 985.4,A -85,B 0,C 180,E1 5980.444,E2 5980.444} C_VEL
LIN {X 0,Y 148.082,Z 976.059,A -85,B 0,C 180,E1 5973.154,E2 5973.154} C_VEL
LIN {X 0,Y 162.588,Z 964.73,A -85,B 0,C 180,E1 5966.941,E2 5966.941} C_VEL
LIN {X 0,Y 176.803,Z 952.769,A -85,B 0,C 180,E1 5962.264,E2 5962.264} C_VEL
LIN {X 0,Y 191.676,Z 939.076,A -85,B 0,C 180,E1 5958.343,E2 5958.343} C_VEL
LIN {X 0,Y 206.411,Z 924.217,A -85,B 0,C 180,E1 5955.162,E2 5955.162} C_VEL
LIN {X 0,Y 220.806,Z 907.893,A -85,B 0,C 180,E1 5952.553,E2 5952.553} C_VEL
LIN {X 0,Y 234.773,Z 890.29,A -85,B 0,C 180,E1 5950.384,E2 5950.384} C_VEL
LIN {X 0,Y 247.305,Z 872.316,A -85,B 0,C 180,E1 5948.682,E2 5948.682} C_VEL
LIN {X 0,Y 260.425,Z 850.889,A -85,B 0,C 180,E1 5947.11,E2 5947.11} C_VEL
LIN {X 0,Y 271.628,Z 829.749,A -85,B 0,C 180,E1 5945.915,E2 5945.915} C_VEL
LIN {X 0,Y 280.989,Z 808.691,A -85,B 0,C 180,E1 5945.003,E2 5945.003} C_VEL
LIN {X 0,Y 289.705,Z 785.379,A -85,B 0,C 180,E1 5944.227,E2 5944.227} C_VEL
LIN {X 0,Y 296.373,Z 763.193,A -85,B 0,C 180,E1 5943.686,E2 5943.686} C_VEL
LIN {X 0,Y 301.807,Z 739.227,A -85,B 0,C 180,E1 5943.222,E2 5943.222} C_VEL
LIN {X 0,Y 305.581,Z 715.087,A -85,B 0,C 180,E1 5942.8,E2 5942.8} C_VEL
LIN {X 0,Y 316.248,Z 626.951,A -85,B 0,C 180,E1 5941.358,E2 5941.358} C_VEL
LIN {X 0,Y 314.439,Z 623.691,A -85,B 0,C 180,E1 5939.088,E2 5939.088} C_VEL
LIN {X 0,Y 312.766,Z 620.524,A -85,B 0,C 180,E1 5936.517,E2 5936.517} C_VEL
LIN {X 0,Y 310.731,Z 616.558,A -85,B 0,C 180,E1 5932.046,E2 5932.046} C_VEL
LIN {X 0,Y 309.57,Z 615.259,A -85,B 0,C 180,E1 5925.981,E2 5925.981} C_VEL
LIN {X 0,Y 310.146,Z 616.049,A -85,B 0,C 180,E1 5920.997,E2 5920.997} C_VEL
LIN {X 0,Y 310.992,Z 616.943,A -85,B 0,C 180,E1 5918.498,E2 5918.498} C_VEL
LIN {X 0,Y 313.48,Z 621.753,A -85,B 0,C 180,E1 5913.59,E2 5913.59} C_VEL
LIN {X 0,Y 315.834,Z 626.142,A -85,B 0,C 180,E1 5910.405,E2 5910.405} C_VEL
LIN {X 0,Y 316.014,Z 626.748,A -85,B 0,C 180,E1 5910.157,E2 5910.157} C_VEL
LIN {X 0,Y 303.97,Z 723.658,A -85,B 0,C 180,E1 5908.6,E2 5908.6} C_VEL
LIN {X 0,Y 299.311,Z 747.229,A -85,B 0,C 180,E1 5908.148,E2 5908.148} C_VEL
LIN {X 0,Y 293.398,Z 769.762,A -85,B 0,C 180,E1 5907.582,E2 5907.582} C_VEL
LIN {X 0,Y 285.961,Z 791.799,A -85,B 0,C 180,E1 5906.853,E2 5906.853} C_VEL
LIN {X 0,Y 276.559,Z 814.773,A -85,B 0,C 180,E1 5905.871,E2 5905.871} C_VEL
LIN {X 0,Y 266.779,Z 834.947,A -85,B 0,C 180,E1 5904.775,E2 5904.775} C_VEL
LIN {X 0,Y 255.314,Z 855.129,A -85,B 0,C 180,E1 5903.386,E2 5903.386} C_VEL
LIN {X 0,Y 242.699,Z 874.602,A -85,B 0,C 180,E1 5901.689,E2 5901.689} C_VEL
LIN {X 0,Y 229.849,Z 891.899,A -85,B 0,C 180,E1 5899.754,E2 5899.754} C_VEL
LIN {X 0,Y 215.18,Z 909.461,A -85,B 0,C 180,E1 5897.222,E2 5897.222} C_VEL
LIN {X 0,Y 201.319,Z 924.269,A -85,B 0,C 180,E1 5894.435,E2 5894.435} C_VEL
LIN {X 0,Y 186.377,Z 938.598,A -85,B 0,C 180,E1 5890.867,E2 5890.867} C_VEL
LIN {X 0,Y 171.443,Z 951.682,A -85,B 0,C 180,E1 5886.489,E2 5886.489} C_VEL
LIN {X 0,Y 157.531,Z 962.691,A -85,B 0,C 180,E1 5881.349,E2 5881.349} C_VEL
LIN {X 0,Y 144.317,Z 972.567,A -85,B 0,C 180,E1 5874.986,E2 5874.986} C_VEL
LIN {X 0,Y 132.898,Z 980.635,A -85,B 0,C 180,E1 5867.5,E2 5867.5} C_VEL
LIN {X 0,Y 122.967,Z 987.744,A -85,B 0,C 180,E1 5857.931,E2 5857.931} C_VEL
LIN {X 0,Y 116.881,Z 992.461,A -85,B 0,C 180,E1 5848.515,E2 5848.515} C_VEL
LIN {X 0,Y 113.258,Z 996.043,A -85,B 0,C 180,E1 5837.752,E2 5837.752} C_VEL
LIN {X 0,Y 112.227,Z 997.785,A -85,B 0,C 180,E1 5829.107,E2 5829.107} C_VEL
LIN {X 0,Y 112.106,Z 998.654,A -85,B 0,C 180,E1 5821.192,E2 5821.192} C_VEL
LIN {X 0,Y 112.386,Z 998.854,A -85,B 0,C 180,E1 5813.2,E2 5813.2} C_VEL
LIN {X 0,Y 113.975,Z 998.24,A -85,B 0,C 180,E1 5803.874,E2 5803.874} C_VEL
LIN {X 0,Y 118.863,Z 996.185,A -85,B 0,C 180,E1 5792.574,E2 5792.574} C_VEL
LIN {X 0,Y 126.809,Z 992.761,A -85,B 0,C 180,E1 5782.674,E2 5782.674} C_VEL
LIN {X 0,Y 139.579,Z 987.178,A -85,B 0,C 180,E1 5772.832,E2 5772.832} C_VEL
LIN {X 0,Y 154.618,Z 980.161,A -85,B 0,C 180,E1 5765.116,E2 5765.116} C_VEL
LIN {X 0,Y 172.04,Z 971.194,A -85,B 0,C 180,E1 5758.746,E2 5758.746} C_VEL
LIN {X 0,Y 190.808,Z 960.595,A -85,B 0,C 180,E1 5753.683,E2 5753.683} C_VEL
LIN {X 0,Y 209.351,Z 948.862,A -85,B 0,C 180,E1 5749.823,E2 5749.823} C_VEL
LIN {X 0,Y 227.037,Z 936.436,A -85,B 0,C 180,E1 5746.837,E2 5746.837} C_VEL
LIN {X 0,Y 207.365,Z 950.878,A -85,B 0,C 180,E1 5743.665,E2 5743.665} C_VEL
LIN {X 0,Y 188.616,Z 963.412,A -85,B 0,C 180,E1 5739.785,E2 5739.785} C_VEL
LIN {X 0,Y 170.203,Z 974.516,A -85,B 0,C 180,E1 5734.799,E2 5734.799} C_VEL
LIN {X 0,Y 160.328,Z 980.138,A -85,B 0,C 180,E1 5731.417,E2 5731.417} C_VEL
LIN {X 0,Y 154.72,Z 983.04,A -85,B 0,C 180,E1 5729.747,E2 5729.747} C_VEL
LIN {X 0,Y 138.542,Z 989.737,A -85,B 0,C 180,E1 5725.87,E2 5725.87} C_VEL
LIN {X 0,Y 133.295,Z 991.976,A -85,B 0,C 180,E1 5723.666,E2 5723.666} C_VEL
LIN {X 0,Y 119.366,Z 998.472,A -85,B 0,C 180,E1 5713.4,E2 5713.4} C_VEL
LIN {X 0,Y 110.114,Z 1002.992,A -85,B 0,C 180,E1 5701.797,E2 5701.797} C_VEL
LIN {X 0,Y 105.403,Z 1005.518,A -85,B 0,C 180,E1 5689.985,E2 5689.985} C_VEL
LIN {X 0,Y 104.107,Z 1006.576,A -85,B 0,C 180,E1 5679.972,E2 5679.972} C_VEL
LIN {X 0,Y 104.086,Z 1006.693,A -85,B 0,C 180,E1 5672.219,E2 5672.219} C_VEL
LIN {X 0,Y 104.072,Z 1006.271,A -85,B 0,C 180,E1 5665.609,E2 5665.609} C_VEL
LIN {X 0,Y 104.286,Z 1005.011,A -85,B 0,C 180,E1 5657.278,E2 5657.278} C_VEL
LIN {X 0,Y 106.147,Z 1002.467,A -85,B 0,C 180,E1 5647.3,E2 5647.3} C_VEL
LIN {X 0,Y 111.666,Z 997.75,A -85,B 0,C 180,E1 5635.46,E2 5635.46} C_VEL
LIN {X 0,Y 119.732,Z 991.911,A -85,B 0,C 180,E1 5625.901,E2 5625.901} C_VEL
LIN {X 0,Y 131.959,Z 983.472,A -85,B 0,C 180,E1 5616.592,E2 5616.592} C_VEL
LIN {X 0,Y 144.999,Z 974.259,A -85,B 0,C 180,E1 5609.703,E2 5609.703} C_VEL
LIN {X 0,Y 159.699,Z 963.145,A -85,B 0,C 180,E1 5603.955,E2 5603.955} C_VEL
LIN {X 0,Y 174.949,Z 950.73,A -85,B 0,C 180,E1 5599.357,E2 5599.357} C_VEL
LIN {X 0,Y 190.042,Z 937.001,A -85,B 0,C 180,E1 5595.717,E2 5595.717} C_VEL
LIN {X 0,Y 205.889,Z 921.128,A -85,B 0,C 180,E1 5592.596,E2 5592.596} C_VEL
LIN {X 0,Y 219.953,Z 905.32,A -85,B 0,C 180,E1 5590.268,E2 5590.268} C_VEL
LIN {X 0,Y 234.771,Z 886.547,A -85,B 0,C 180,E1 5588.162,E2 5588.162} C_VEL
LIN {X 0,Y 247.557,Z 868.244,A -85,B 0,C 180,E1 5586.583,E2 5586.583} C_VEL
LIN {X 0,Y 259.47,Z 848.524,A -85,B 0,C 180,E1 5585.271,E2 5585.271} C_VEL
LIN {X 0,Y 270.637,Z 827.31,A -85,B 0,C 180,E1 5584.17,E2 5584.17} C_VEL
LIN {X 0,Y 279.806,Z 806.701,A -85,B 0,C 180,E1 5583.345,E2 5583.345} C_VEL
LIN {X 0,Y 288.471,Z 783.324,A -85,B 0,C 180,E1 5582.631,E2 5582.631} C_VEL
LIN {X 0,Y 295.398,Z 760.196,A -85,B 0,C 180,E1 5582.114,E2 5582.114} C_VEL
LIN {X 0,Y 300.565,Z 736.645,A -85,B 0,C 180,E1 5581.688,E2 5581.688} C_VEL
LIN {X 0,Y 304.903,Z 707.119,A -85,B 0,C 180,E1 5581.2,E2 5581.2} C_VEL
LIN {X 0,Y 314.068,Z 633.008,A -85,B 0,C 180,E1 5580.04,E2 5580.04} C_VEL
LIN {X 0,Y 311.534,Z 628.355,A -85,B 0,C 180,E1 5576.319,E2 5576.319} C_VEL
LIN {X 0,Y 309.628,Z 624.483,A -85,B 0,C 180,E1 5572.018,E2 5572.018} C_VEL
LIN {X 0,Y 308.478,Z 623.182,A -85,B 0,C 180,E1 5565.93,E2 5565.93} C_VEL
LIN {X 0,Y 309.132,Z 624.043,A -85,B 0,C 180,E1 5560.736,E2 5560.736} C_VEL
LIN {X 0,Y 309.84,Z 624.885,A -85,B 0,C 180,E1 5558.613,E2 5558.613} C_VEL
LIN {X 0,Y 312.184,Z 629.502,A -85,B 0,C 180,E1 5553.871,E2 5553.871} C_VEL
LIN {X 0,Y 313.84,Z 632.657,A -85,B 0,C 180,E1 5551.5,E2 5551.5} C_VEL
LIN {X 0,Y 302.25,Z 724.072,A -85,B 0,C 180,E1 5550.075,E2 5550.075} C_VEL
LIN {X 0,Y 297.498,Z 747.727,A -85,B 0,C 180,E1 5549.641,E2 5549.641} C_VEL
LIN {X 0,Y 291.54,Z 770.13,A -85,B 0,C 180,E1 5549.105,E2 5549.105} C_VEL
LIN {X 0,Y 284.459,Z 790.964,A -85,B 0,C 180,E1 5548.456,E2 5548.456} C_VEL
LIN {X 0,Y 275.379,Z 813.235,A -85,B 0,C 180,E1 5547.568,E2 5547.568} C_VEL
LIN {X 0,Y 265.502,Z 833.527,A -85,B 0,C 180,E1 5546.537,E2 5546.537} C_VEL
LIN {X 0,Y 253.791,Z 854.138,A -85,B 0,C 180,E1 5545.212,E2 5545.212} C_VEL
LIN {X 0,Y 241.335,Z 873.244,A -85,B 0,C 180,E1 5543.654,E2 5543.654} C_VEL
LIN {X 0,Y 227.658,Z 891.426,A -85,B 0,C 180,E1 5541.736,E2 5541.736} C_VEL
LIN {X 0,Y 213.23,Z 908.508,A -85,B 0,C 180,E1 5539.417,E2 5539.417} C_VEL
LIN {X 0,Y 198.98,Z 923.458,A -85,B 0,C 180,E1 5536.755,E2 5536.755} C_VEL
LIN {X 0,Y 182.769,Z 938.699,A -85,B 0,C 180,E1 5533.128,E2 5533.128} C_VEL
LIN {X 0,Y 168.048,Z 951.183,A -85,B 0,C 180,E1 5529.085,E2 5529.085} C_VEL
LIN {X 0,Y 153.475,Z 962.339,A -85,B 0,C 180,E1 5524.059,E2 5524.059} C_VEL
LIN {X 0,Y 139.498,Z 972.364,A -85,B 0,C 180,E1 5517.752,E2 5517.752} C_VEL
LIN {X 0,Y 126.729,Z 980.867,A -85,B 0,C 180,E1 5509.816,E2 5509.816} C_VEL
LIN {X 0,Y 116.025,Z 988.004,A -85,B 0,C 180,E1 5499.909,E2 5499.909} C_VEL
LIN {X 0,Y 109.377,Z 992.73,A -85,B 0,C 180,E1 5489.984,E2 5489.984} C_VEL
LIN {X 0,Y 105.277,Z 996.422,A -85,B 0,C 180,E1 5478.033,E2 5478.033} C_VEL
LIN {X 0,Y 104.202,Z 998.16,A -85,B 0,C 180,E1 5468.559,E2 5468.559} C_VEL
LIN {X 0,Y 104.108,Z 998.96,A -85,B 0,C 180,E1 5460.654,E2 5460.654} C_VEL
LIN {X 0,Y 104.471,Z 999.177,A -85,B 0,C 180,E1 5452.209,E2 5452.209} C_VEL
LIN {X 0,Y 106.419,Z 998.582,A -85,B 0,C 180,E1 5442.056,E2 5442.056} C_VEL
LIN {X 0,Y 112.179,Z 996.534,A -85,B 0,C 180,E1 5429.945,E2 5429.945} C_VEL
LIN {X 0,Y 121.735,Z 992.902,A -85,B 0,C 180,E1 5419.135,E2 5419.135} C_VEL
LIN {X 0,Y 135.876,Z 987.261,A -85,B 0,C 180,E1 5409.318,E2 5409.318} C_VEL
LIN {X 0,Y 152.078,Z 980.246,A -85,B 0,C 180,E1 5401.807,E2 5401.807} C_VEL
LIN {X 0,Y 170.471,Z 971.275,A -85,B 0,C 180,E1 5395.737,E2 5395.737} C_VEL
LIN {X 0,Y 190.205,Z 960.59,A -85,B 0,C 180,E1 5390.928,E2 5390.928} C_VEL
LIN {X 0,Y 209.51,Z 948.82,A -85,B 0,C 180,E1 5387.32,E2 5387.32} C_VEL
LIN {X 0,Y 212.001,Z 947.252,A -85,B 0,C 180,E1 5386.917,E2 5386.917} C_VEL
LIN {X 0,Y 192.855,Z 959.728,A -85,B 0,C 180,E1 5383.588,E2 5383.588} C_VEL
LIN {X 0,Y 173.341,Z 971.364,A -85,B 0,C 180,E1 5379.16,E2 5379.16} C_VEL
LIN {X 0,Y 155.929,Z 980.746,A -85,B 0,C 180,E1 5373.88,E2 5373.88} C_VEL
LIN {X 0,Y 138.17,Z 989.638,A -85,B 0,C 180,E1 5366.344,E2 5366.344} C_VEL
LIN {X 0,Y 133.295,Z 991.976,A -85,B 0,C 180,E1 5363.666,E2 5363.666} C_VEL
LIN {X 0,Y 128.211,Z 994.13,A -85,B 0,C 180,E1 5361.269,E2 5361.269} C_VEL
LIN {X 0,Y 112.667,Z 999.116,A -85,B 0,C 180,E1 5354.773,E2 5354.773} C_VEL
LIN {X 0,Y 109.038,Z 1000.324,A -85,B 0,C 180,E1 5351.949,E2 5351.949} C_VEL
LIN {X 0,Y 100.727,Z 1003.842,A -85,B 0,C 180,E1 5339.776,E2 5339.776} C_VEL
LIN {X 0,Y 96.747,Z 1005.927,A -85,B 0,C 180,E1 5326.839,E2 5326.839} C_VEL
LIN {X 0,Y 96.055,Z 1006.444,A -85,B 0,C 180,E1 5315.993,E2 5315.993} C_VEL
LIN {X 0,Y 96.103,Z 1006.222,A -85,B 0,C 180,E1 5308.23,E2 5308.23} C_VEL
LIN {X 0,Y 96.16,Z 1005.172,A -85,B 0,C 180,E1 5299.232,E2 5299.232} C_VEL
LIN {X 0,Y 97.894,Z 1002.66,A -85,B 0,C 180,E1 5287.816,E2 5287.816} C_VEL
LIN {X 0,Y 102.709,Z 998.731,A -85,B 0,C 180,E1 5276.319,E2 5276.319} C_VEL
LIN {X 0,Y 111.661,Z 992.661,A -85,B 0,C 180,E1 5265.001,E2 5265.001} C_VEL
LIN {X 0,Y 123.315,Z 985.232,A -85,B 0,C 180,E1 5255.852,E2 5255.852} C_VEL
LIN {X 0,Y 136.651,Z 976.327,A -85,B 0,C 180,E1 5248.626,E2 5248.626} C_VEL
LIN {X 0,Y 151.679,Z 965.773,A -85,B 0,C 180,E1 5242.685,E2 5242.685} C_VEL
LIN {X 0,Y 167.143,Z 953.742,A -85,B 0,C 180,E1 5238.024,E2 5238.024} C_VEL
LIN {X 0,Y 183.496,Z 939.784,A -85,B 0,C 180,E1 5234.139,E2 5234.139} C_VEL
LIN {X 0,Y 197.812,Z 926.162,A -85,B 0,C 180,E1 5231.363,E2 5231.363} C_VEL
LIN {X 0,Y 213.924,Z 909.003,A -85,B 0,C 180,E1 5228.755,E2 5228.755} C_VEL
LIN {X 0,Y 228.196,Z 891.895,A -85,B 0,C 180,E1 5226.793,E2 5226.793} C_VEL
LIN {X 0,Y 241.904,Z 873.084,A -85,B 0,C 180,E1 5225.155,E2 5225.155} C_VEL
LIN {X 0,Y 254.531,Z 853.436,A -85,B 0,C 180,E1 5223.828,E2 5223.828} C_VEL
LIN {X 0,Y 265.335,Z 833.906,A -85,B 0,C 180,E1 5222.807,E2 5222.807} C_VEL
LIN {X 0,Y 276.07,Z 811.24,A -85,B 0,C 180,E1 5221.893,E2 5221.893} C_VEL
LIN {X 0,Y 284.534,Z 789.895,A -85,B 0,C 180,E1 5221.236,E2 5221.236} C_VEL
LIN {X 0,Y 291.877,Z 766.872,A -85,B 0,C 180,E1 5220.717,E2 5220.717} C_VEL
LIN {X 0,Y 297.715,Z 743.4,A -85,B 0,C 180,E1 5220.298,E2 5220.298} C_VEL
LIN {X 0,Y 301.675,Z 720.364,A -85,B 0,C 180,E1 5219.922,E2 5219.922} C_VEL
LIN {X 0,Y 311.882,Z 639.341,A -85,B 0,C 180,E1 5218.667,E2 5218.667} C_VEL
LIN {X 0,Y 310.194,Z 636.035,A -85,B 0,C 180,E1 5215.933,E2 5215.933} C_VEL
LIN {X 0,Y 308.459,Z 632.352,A -85,B 0,C 180,E1 5211.799,E2 5211.799} C_VEL
LIN {X 0,Y 307.378,Z 631.099,A -85,B 0,C 180,E1 5205.747,E2 5205.747} C_VEL
LIN {X 0,Y 308.225,Z 632.114,A -85,B 0,C 180,E1 5200.153,E2 5200.153} C_VEL
LIN {X 0,Y 308.689,Z 632.825,A -85,B 0,C 180,E1 5198.729,E2 5198.729} C_VEL
LIN {X 0,Y 310.945,Z 637.37,A -85,B 0,C 180,E1 5194.067,E2 5194.067} C_VEL
LIN {X 0,Y 311.688,Z 639.188,A -85,B 0,C 180,E1 5192.849,E2 5192.849} C_VEL
LIN {X 0,Y 300.703,Z 724.581,A -85,B 0,C 180,E1 5191.563,E2 5191.563} C_VEL
LIN {X 0,Y 295.892,Z 748.178,A -85,B 0,C 180,E1 5191.152,E2 5191.152} C_VEL
LIN {X 0,Y 289.889,Z 770.453,A -85,B 0,C 180,E1 5190.648,E2 5190.648} C_VEL
LIN {X 0,Y 282.719,Z 791.278,A -85,B 0,C 180,E1 5190.034,E2 5190.034} C_VEL
LIN {X 0,Y 273.519,Z 813.541,A -85,B 0,C 180,E1 5189.194,E2 5189.194} C_VEL
LIN {X 0,Y 263.902,Z 833.065,A -85,B 0,C 180,E1 5188.258,E2 5188.258} C_VEL
LIN {X 0,Y 251.615,Z 854.447,A -85,B 0,C 180,E1 5186.962,E2 5186.962} C_VEL
LIN {X 0,Y 238.998,Z 873.53,A -85,B 0,C 180,E1 5185.487,E2 5185.487} C_VEL
LIN {X 0,Y 225.191,Z 891.602,A -85,B 0,C 180,E1 5183.678,E2 5183.678} C_VEL
LIN {X 0,Y 210.73,Z 908.451,A -85,B 0,C 180,E1 5181.509,E2 5181.509} C_VEL
LIN {X 0,Y 196.127,Z 923.437,A -85,B 0,C 180,E1 5178.966,E2 5178.966} C_VEL
LIN {X 0,Y 179.45,Z 938.731,A -85,B 0,C 180,E1 5175.479,E2 5175.479} C_VEL
LIN {X 0,Y 164.226,Z 951.264,A -85,B 0,C 180,E1 5171.561,E2 5171.561} C_VEL
LIN {X 0,Y 149.045,Z 962.485,A -85,B 0,C 180,E1 5166.643,E2 5166.643} C_VEL
LIN {X 0,Y 134.361,Z 972.551,A -85,B 0,C 180,E1 5160.383,E2 5160.383} C_VEL
LIN {X 0,Y 120.784,Z 981.075,A -85,B 0,C 180,E1 5152.366,E2 5152.366} C_VEL
LIN {X 0,Y 109.232,Z 988.237,A -85,B 0,C 180,E1 5142.137,E2 5142.137} C_VEL
LIN {X 0,Y 101.952,Z 992.98,A -85,B 0,C 180,E1 5131.669,E2 5131.669} C_VEL
LIN {X 0,Y 97.501,Z 996.6,A -85,B 0,C 180,E1 5119.345,E2 5119.345} C_VEL
LIN {X 0,Y 96.237,Z 998.369,A -85,B 0,C 180,E1 5109.244,E2 5109.244} C_VEL
LIN {X 0,Y 96.114,Z 999.227,A -85,B 0,C 180,E1 5100.71,E2 5100.71} C_VEL
LIN {X 0,Y 96.528,Z 999.511,A -85,B 0,C 180,E1 5091.554,E2 5091.554} C_VEL
LIN {X 0,Y 98.771,Z 998.985,A -85,B 0,C 180,E1 5080.58,E2 5080.58} C_VEL
LIN {X 0,Y 105.204,Z 997.097,A -85,B 0,C 180,E1 5067.758,E2 5067.758} C_VEL
LIN {X 0,Y 115.75,Z 993.535,A -85,B 0,C 180,E1 5056.453,E2 5056.453} C_VEL
LIN {X 0,Y 130.867,Z 988.106,A -85,B 0,C 180,E1 5046.574,E2 5046.574} C_VEL
LIN {X 0,Y 147.009,Z 981.608,A -85,B 0,C 180,E1 5039.492,E2 5039.492} C_VEL
LIN {X 0,Y 166.422,Z 972.845,A -85,B 0,C 180,E1 5033.447,E2 5033.447} C_VEL
LIN {X 0,Y 185.347,Z 963.258,A -85,B 0,C 180,E1 5029.091,E2 5029.091} C_VEL
LIN {X 0,Y 196.49,Z 957.018,A -85,B 0,C 180,E1 5026.945,E2 5026.945} C_VEL
LIN {X 0,Y 177.326,Z 968.179,A -85,B 0,C 180,E1 5023.289,E2 5023.289} C_VEL
LIN {X 0,Y 156.455,Z 979.105,A -85,B 0,C 180,E1 5017.943,E2 5017.943} C_VEL
LIN {X 0,Y 138.007,Z 987.927,A -85,B 0,C 180,E1 5011.262,E2 5011.262} C_VEL
LIN {X 0,Y 121.313,Z 995.138,A -85,B 0,C 180,E1 5002.321,E2 5002.321} C_VEL
LIN {X 0,Y 109.038,Z 1000.324,A -85,B 0,C 180,E1 4991.949,E2 4991.949} C_VEL
LIN {X 0,Y 105.016,Z 1001.614,A -85,B 0,C 180,E1 4988.455,E2 4988.455} C_VEL
LIN {X 0,Y 95.835,Z 1003.715,A -85,B 0,C 180,E1 4981.692,E2 4981.692} C_VEL
LIN {X 0,Y 91.369,Z 1004.662,A -85,B 0,C 180,E1 4976.59,E2 4976.59} C_VEL
LIN {X 0,Y 90.473,Z 1004.921,A -85,B 0,C 180,E1 4974.568,E2 4974.568} C_VEL
LIN {X 0,Y 88.229,Z 1005.976,A -85,B 0,C 180,E1 4962.454,E2 4962.454} C_VEL
LIN {X 0,Y 88.086,Z 1006.044,A -85,B 0,C 180,E1 4952.768,E2 4952.768} C_VEL
LIN {X 0,Y 88.083,Z 1005.591,A -85,B 0,C 180,E1 4945.463,E2 4945.463} C_VEL
LIN {X 0,Y 88.424,Z 1004.278,A -85,B 0,C 180,E1 4935.616,E2 4935.616} C_VEL
LIN {X 0,Y 90.948,Z 1001.675,A -85,B 0,C 180,E1 4923.935,E2 4923.935} C_VEL
LIN {X 0,Y 97.844,Z 996.921,A -85,B 0,C 180,E1 4910.711,E2 4910.711} C_VEL
LIN {X 0,Y 107.551,Z 991.026,A -85,B 0,C 180,E1 4900.359,E2 4900.359} C_VEL
LIN {X 0,Y 121.277,Z 982.74,A -85,B 0,C 180,E1 4891.004,E2 4891.004} C_VEL
LIN {X 0,Y 135.86,Z 973.487,A -85,B 0,C 180,E1 4884.173,E2 4884.173} C_VEL
LIN {X 0,Y 151.927,Z 962.296,A -85,B 0,C 180,E1 4878.657,E2 4878.657} C_VEL
LIN {X 0,Y 168.213,Z 949.868,A -85,B 0,C 180,E1 4874.384,E2 4874.384} C_VEL
LIN {X 0,Y 184.34,Z 935.975,A -85,B 0,C 180,E1 4871.026,E2 4871.026} C_VEL
LIN {X 0,Y 201.459,Z 919.48,A -85,B 0,C 180,E1 4868.133,E2 4868.133} C_VEL
LIN {X 0,Y 216.139,Z 903.536,A -85,B 0,C 180,E1 4866.06,E2 4866.06} C_VEL
LIN {X 0,Y 230.579,Z 885.711,A -85,B 0,C 180,E1 4864.306,E2 4864.306} C_VEL
LIN {X 0,Y 243.905,Z 867.133,A -85,B 0,C 180,E1 4862.899,E2 4862.899} C_VEL
LIN {X 0,Y 256.044,Z 847.466,A -85,B 0,C 180,E1 4861.759,E2 4861.759} C_VEL
LIN {X 0,Y 267.447,Z 826.195,A -85,B 0,C 180,E1 4860.802,E2 4860.802} C_VEL
LIN {X 0,Y 276.42,Z 806.448,A -85,B 0,C 180,E1 4860.115,E2 4860.115} C_VEL
LIN {X 0,Y 285.429,Z 782.634,A -85,B 0,C 180,E1 4859.484,E2 4859.484} C_VEL
LIN {X 0,Y 292.458,Z 759.558,A -85,B 0,C 180,E1 4859.041,E2 4859.041} C_VEL
LIN {X 0,Y 297.716,Z 736.009,A -85,B 0,C 180,E1 4858.661,E2 4858.661} C_VEL
LIN {X 0,Y 302.283,Z 705.536,A -85,B 0,C 180,E1 4858.198,E2 4858.198} C_VEL
LIN {X 0,Y 309.895,Z 645.728,A -85,B 0,C 180,E1 4857.318,E2 4857.318} C_VEL
LIN {X 0,Y 308.856,Z 643.701,A -85,B 0,C 180,E1 4855.524,E2 4855.524} C_VEL
LIN {X 0,Y 307.269,Z 640.202,A -85,B 0,C 180,E1 4851.526,E2 4851.526} C_VEL
LIN {X 0,Y 306.28,Z 639.02,A -85,B 0,C 180,E1 4845.634,E2 4845.634} C_VEL
LIN {X 0,Y 307.171,Z 640.084,A -85,B 0,C 180,E1 4840.014,E2 4840.014} C_VEL
LIN {X 0,Y 307.601,Z 640.963,A -85,B 0,C 180,E1 4838.65,E2 4838.65} C_VEL
LIN {X 0,Y 309.655,Z 645.105,A -85,B 0,C 180,E1 4834.361,E2 4834.361} C_VEL
LIN {X 0,Y 309.707,Z 645.491,A -85,B 0,C 180,E1 4834.218,E2 4834.218} C_VEL
LIN {X 0,Y 299.292,Z 724.944,A -85,B 0,C 180,E1 4833.066,E2 4833.066} C_VEL
LIN {X 0,Y 294.425,Z 748.498,A -85,B 0,C 180,E1 4832.678,E2 4832.678} C_VEL
LIN {X 0,Y 288.208,Z 771.221,A -85,B 0,C 180,E1 4832.191,E2 4832.191} C_VEL
LIN {X 0,Y 280.726,Z 792.638,A -85,B 0,C 180,E1 4831.593,E2 4831.593} C_VEL
LIN {X 0,Y 270.948,Z 815.693,A -85,B 0,C 180,E1 4830.761,E2 4830.761} C_VEL
LIN {X 0,Y 260.751,Z 835.947,A -85,B 0,C 180,E1 4829.83,E2 4829.83} C_VEL
LIN {X 0,Y 248.757,Z 856.186,A -85,B 0,C 180,E1 4828.646,E2 4828.646} C_VEL
LIN {X 0,Y 235.95,Z 875.077,A -85,B 0,C 180,E1 4827.246,E2 4827.246} C_VEL
LIN {X 0,Y 221.914,Z 893.004,A -85,B 0,C 180,E1 4825.523,E2 4825.523} C_VEL
LIN {X 0,Y 205.854,Z 911.051,A -85,B 0,C 180,E1 4823.249,E2 4823.249} C_VEL
LIN {X 0,Y 190.117,Z 926.709,A -85,B 0,C 180,E1 4820.616,E2 4820.616} C_VEL
LIN {X 0,Y 173.92,Z 940.84,A -85,B 0,C 180,E1 4817.363,E2 4817.363} C_VEL
LIN {X 0,Y 157.489,Z 953.734,A -85,B 0,C 180,E1 4813.27,E2 4813.27} C_VEL
LIN {X 0,Y 141.904,Z 964.651,A -85,B 0,C 180,E1 4808.302,E2 4808.302} C_VEL
LIN {X 0,Y 126.069,Z 974.743,A -85,B 0,C 180,E1 4801.546,E2 4801.546} C_VEL
LIN {X 0,Y 112.715,Z 982.687,A -85,B 0,C 180,E1 4793.509,E2 4793.509} C_VEL
LIN {X 0,Y 101.239,Z 989.24,A -85,B 0,C 180,E1 4783.111,E2 4783.111} C_VEL
LIN {X 0,Y 93.393,Z 994.08,A -85,B 0,C 180,E1 4771.208,E2 4771.208} C_VEL
LIN {X 0,Y 89.251,Z 997.234,A -85,B 0,C 180,E1 4758.347,E2 4758.347} C_VEL
LIN {X 0,Y 88.181,Z 998.805,A -85,B 0,C 180,E1 4748.006,E2 4748.006} C_VEL
LIN {X 0,Y 88.126,Z 999.564,A -85,B 0,C 180,E1 4739.277,E2 4739.277} C_VEL
LIN {X 0,Y 88.818,Z 999.817,A -85,B 0,C 180,E1 4728.963,E2 4728.963} C_VEL
LIN {X 0,Y 92.018,Z 999.214,A -85,B 0,C 180,E1 4716.703,E2 4716.703} C_VEL
LIN {X 0,Y 100.91,Z 996.878,A -85,B 0,C 180,E1 4702.121,E2 4702.121} C_VEL
LIN {X 0,Y 113.167,Z 993.253,A -85,B 0,C 180,E1 4691.204,E2 4691.204} C_VEL
LIN {X 0,Y 130.15,Z 987.519,A -85,B 0,C 180,E1 4681.763,E2 4681.763} C_VEL
LIN {X 0,Y 148.583,Z 980.531,A -85,B 0,C 180,E1 4674.936,E2 4674.936} C_VEL
LIN {X 0,Y 168.772,Z 971.606,A -85,B 0,C 180,E1 4669.601,E2 4669.601} C_VEL
LIN {X 0,Y 181.17,Z 965.567,A -85,B 0,C 180,E1 4667.01,E2 4667.01} C_VEL
LIN {X 0,Y 160.353,Z 976.339,A -85,B 0,C 180,E1 4662.585,E2 4662.585} C_VEL
LIN {X 0,Y 140.436,Z 985.391,A -85,B 0,C 180,E1 4656.725,E2 4656.725} C_VEL
LIN {X 0,Y 121.781,Z 993.125,A -85,B 0,C 180,E1 4648.659,E2 4648.659} C_VEL
LIN {X 0,Y 106.749,Z 998.827,A -85,B 0,C 180,E1 4638.553,E2 4638.553} C_VEL
LIN {X 0,Y 95.102,Z 1003.111,A -85,B 0,C 180,E1 4624.914,E2 4624.914} C_VEL
LIN {X 0,Y 90.473,Z 1004.921,A -85,B 0,C 180,E1 4614.568,E2 4614.568} C_VEL
LIN {X 0,Y 88.277,Z 1005.524,A -85,B 0,C 180,E1 4609.806,E2 4609.806} C_VEL
LIN {X 0,Y 83.614,Z 1005.871,A -85,B 0,C 180,E1 4602.199,E2 4602.199} C_VEL
LIN {X 0,Y 80.201,Z 1005.724,A -85,B 0,C 180,E1 4593,E2 4593} C_VEL
LIN {X 0,Y 80.114,Z 1005.685,A -85,B 0,C 180,E1 4591.386,E2 4591.386} C_VEL
LIN {X 0,Y 80.081,Z 1005.01,A -85,B 0,C 180,E1 4582.85,E2 4582.85} C_VEL
LIN {X 0,Y 81.242,Z 1003.131,A -85,B 0,C 180,E1 4569.866,E2 4569.866} C_VEL
LIN {X 0,Y 86.45,Z 999.294,A -85,B 0,C 180,E1 4555.197,E2 4555.197} C_VEL
LIN {X 0,Y 96.012,Z 993.866,A -85,B 0,C 180,E1 4542.35,E2 4542.35} C_VEL
LIN {X 0,Y 108.774,Z 986.708,A -85,B 0,C 180,E1 4532.215,E2 4532.215} C_VEL
LIN {X 0,Y 123.918,Z 977.938,A -85,B 0,C 180,E1 4524.289,E2 4524.289} C_VEL
LIN {X 0,Y 139.205,Z 968.203,A -85,B 0,C 180,E1 4518.586,E2 4518.586} C_VEL
LIN {X 0,Y 157.333,Z 955.459,A -85,B 0,C 180,E1 4513.569,E2 4513.569} C_VEL
LIN {X 0,Y 173.622,Z 942.632,A -85,B 0,C 180,E1 4510.087,E2 4510.087} C_VEL
LIN {X 0,Y 190.433,Z 927.645,A -85,B 0,C 180,E1 4507.191,E2 4507.191} C_VEL
LIN {X 0,Y 206.203,Z 911.92,A -85,B 0,C 180,E1 4504.955,E2 4504.955} C_VEL
LIN {X 0,Y 221.262,Z 894.708,A -85,B 0,C 180,E1 4503.141,E2 4503.141} C_VEL
LIN {X 0,Y 236.515,Z 874.888,A -85,B 0,C 180,E1 4501.566,E2 4501.566} C_VEL
LIN {X 0,Y 249.43,Z 855.633,A -85,B 0,C 180,E1 4500.401,E2 4500.401} C_VEL
LIN {X 0,Y 260.933,Z 835.656,A -85,B 0,C 180,E1 4499.473,E2 4499.473} C_VEL
LIN {X 0,Y 271.489,Z 814.46,A -85,B 0,C 180,E1 4498.71,E2 4498.71} C_VEL
LIN {X 0,Y 280.319,Z 793.018,A -85,B 0,C 180,E1 4498.127,E2 4498.127} C_VEL
LIN {X 0,Y 288.538,Z 768.582,A -85,B 0,C 180,E1 4497.637,E2 4497.637} C_VEL
LIN {X 0,Y 294.611,Z 745.335,A -85,B 0,C 180,E1 4497.274,E2 4497.274} C_VEL
LIN {X 0,Y 298.907,Z 721.574,A -85,B 0,C 180,E1 4496.923,E2 4496.923} C_VEL
LIN {X 0,Y 307.959,Z 651.995,A -85,B 0,C 180,E1 4495.903,E2 4495.903} C_VEL
LIN {X 0,Y 306.108,Z 648.082,A -85,B 0,C 180,E1 4491.358,E2 4491.358} C_VEL
LIN {X 0,Y 305.184,Z 646.944,A -85,B 0,C 180,E1 4485.581,E2 4485.581} C_VEL
LIN {X 0,Y 306.16,Z 648.094,A -85,B 0,C 180,E1 4479.746,E2 4479.746} C_VEL
LIN {X 0,Y 307.799,Z 652.013,A -85,B 0,C 180,E1 4475.601,E2 4475.601} C_VEL
LIN {X 0,Y 298.03,Z 725.534,A -85,B 0,C 180,E1 4474.578,E2 4474.578} C_VEL
LIN {X 0,Y 293.079,Z 749.13,A -85,B 0,C 180,E1 4474.212,E2 4474.212} C_VEL
LIN {X 0,Y 286.738,Z 771.961,A -85,B 0,C 180,E1 4473.752,E2 4473.752} C_VEL
LIN {X 0,Y 279.41,Z 792.7,A -85,B 0,C 180,E1 4473.212,E2 4473.212} C_VEL
LIN {X 0,Y 269.519,Z 815.799,A -85,B 0,C 180,E1 4472.435,E2 4472.435} C_VEL
LIN {X 0,Y 259.196,Z 836.072,A -85,B 0,C 180,E1 4471.566,E2 4471.566} C_VEL
LIN {X 0,Y 247.042,Z 856.339,A -85,B 0,C 180,E1 4470.46,E2 4470.46} C_VEL
LIN {X 0,Y 233.812,Z 875.591,A -85,B 0,C 180,E1 4469.124,E2 4469.124} C_VEL
LIN {X 0,Y 219.828,Z 893.205,A -85,B 0,C 180,E1 4467.539,E2 4467.539} C_VEL
LIN {X 0,Y 203.878,Z 910.886,A -85,B 0,C 180,E1 4465.459,E2 4465.459} C_VEL
LIN {X 0,Y 188.67,Z 925.762,A -85,B 0,C 180,E1 4463.133,E2 4463.133} C_VEL
LIN {X 0,Y 172.03,Z 940.101,A -85,B 0,C 180,E1 4460.085,E2 4460.085} C_VEL
LIN {X 0,Y 155.886,Z 952.593,A -85,B 0,C 180,E1 4456.432,E2 4456.432} C_VEL
LIN {X 0,Y 139.582,Z 963.7,A -85,B 0,C 180,E1 4451.754,E2 4451.754} C_VEL
LIN {X 0,Y 123.558,Z 973.663,A -85,B 0,C 180,E1 4445.617,E2 4445.617} C_VEL
LIN {X 0,Y 109.068,Z 981.788,A -85,B 0,C 180,E1 4437.855,E2 4437.855} C_VEL
LIN {X 0,Y 95.734,Z 988.928,A -85,B 0,C 180,E1 4426.984,E2 4426.984} C_VEL
LIN {X 0,Y 87.07,Z 993.663,A -85,B 0,C 180,E1 4415.251,E2 4415.251} C_VEL
LIN {X 0,Y 81.68,Z 997.25,A -85,B 0,C 180,E1 4400.822,E2 4400.822} C_VEL
LIN {X 0,Y 80.215,Z 999.003,A -85,B 0,C 180,E1 4388.787,E2 4388.787} C_VEL
LIN {X 0,Y 80.132,Z 999.829,A -85,B 0,C 180,E1 4379.207,E2 4379.207} C_VEL
LIN {X 0,Y 80.952,Z 1000.154,A -85,B 0,C 180,E1 4367.827,E2 4367.827} C_VEL
LIN {X 0,Y 84.744,Z 999.612,A -85,B 0,C 180,E1 4354.287,E2 4354.287} C_VEL
LIN {X 0,Y 94.599,Z 997.472,A -85,B 0,C 180,E1 4339.129,E2 4339.129} C_VEL
LIN {X 0,Y 108.038,Z 993.93,A -85,B 0,C 180,E1 4327.907,E2 4327.907} C_VEL
LIN {X 0,Y 127.109,Z 988.073,A -85,B 0,C 180,E1 4318.199,E2 4318.199} C_VEL
LIN {X 0,Y 146.531,Z 981.174,A -85,B 0,C 180,E1 4311.722,E2 4311.722} C_VEL
LIN {X 0,Y 165.657,Z 973.202,A -85,B 0,C 180,E1 4307.047,E2 4307.047} C_VEL
LIN {X 0,Y 143.258,Z 983.27,A -85,B 0,C 180,E1 4301.69,E2 4301.69} C_VEL
LIN {X 0,Y 124.477,Z 990.715,A -85,B 0,C 180,E1 4295.214,E2 4295.214} C_VEL
LIN {X 0,Y 105.817,Z 997.318,A -85,B 0,C 180,E1 4285.317,E2 4285.317} C_VEL
LIN {X 0,Y 91.727,Z 1001.981,A -85,B 0,C 180,E1 4272.542,E2 4272.542} C_VEL
LIN {X 0,Y 83.403,Z 1004.58,A -85,B 0,C 180,E1 4257.897,E2 4257.897} C_VEL
LIN {X 0,Y 80.337,Z 1005.687,A -85,B 0,C 180,E1 4243.898,E2 4243.898} C_VEL
LIN {X 0,Y 80.08,Z 1005.726,A -85,B 0,C 180,E1 4233.601,E2 4233.601} C_VEL
LIN {X 0,Y 80.114,Z 1005.685,A -85,B 0,C 180,E1 4231.386,E2 4231.386} C_VEL
LIN {X 0,Y 79.353,Z 1005.448,A -85,B 0,C 180,E1 4226.666,E2 4226.666} C_VEL
LIN {X 0,Y 76.946,Z 1004.778,A -85,B 0,C 180,E1 4220.374,E2 4220.374} C_VEL
LIN {X 0,Y 73.789,Z 1002.913,A -85,B 0,C 180,E1 4208.976,E2 4208.976} C_VEL
LIN {X 0,Y 74.248,Z 1002.123,A -85,B 0,C 180,E1 4205.074,E2 4205.074} C_VEL
LIN {X 0,Y 80.02,Z 998.586,A -85,B 0,C 180,E1 4191.366,E2 4191.366} C_VEL
LIN {X 0,Y 91.208,Z 992.832,A -85,B 0,C 180,E1 4177.868,E2 4177.868} C_VEL
LIN {X 0,Y 104.475,Z 985.944,A -85,B 0,C 180,E1 4168.341,E2 4168.341} C_VEL
LIN {X 0,Y 121.924,Z 976.255,A -85,B 0,C 180,E1 4160.145,E2 4160.145} C_VEL
LIN {X 0,Y 137.617,Z 966.627,A -85,B 0,C 180,E1 4154.972,E2 4154.972} C_VEL
LIN {X 0,Y 155.561,Z 954.231,A -85,B 0,C 180,E1 4150.529,E2 4150.529} C_VEL
LIN {X 0,Y 172.338,Z 941.279,A -85,B 0,C 180,E1 4147.306,E2 4147.306} C_VEL
LIN {X 0,Y 189.558,Z 926.063,A -85,B 0,C 180,E1 4144.646,E2 4144.646} C_VEL
LIN {X 0,Y 206.564,Z 909.081,A -85,B 0,C 180,E1 4142.496,E2 4142.496} C_VEL
LIN {X 0,Y 220.96,Z 892.72,A -85,B 0,C 180,E1 4140.949,E2 4140.949} C_VEL
LIN {X 0,Y 235.604,Z 873.685,A -85,B 0,C 180,E1 4139.589,E2 4139.589} C_VEL
LIN {X 0,Y 248.505,Z 854.568,A -85,B 0,C 180,E1 4138.539,E2 4138.539} C_VEL
LIN {X 0,Y 260.133,Z 834.378,A -85,B 0,C 180,E1 4137.692,E2 4137.692} C_VEL
LIN {X 0,Y 270.792,Z 812.888,A -85,B 0,C 180,E1 4136.997,E2 4136.997} C_VEL
LIN {X 0,Y 279.7,Z 791.278,A -85,B 0,C 180,E1 4136.468,E2 4136.468} C_VEL
LIN {X 0,Y 287.668,Z 767.452,A -85,B 0,C 180,E1 4136.045,E2 4136.045} C_VEL
LIN {X 0,Y 293.77,Z 744.035,A -85,B 0,C 180,E1 4135.711,E2 4135.711} C_VEL
LIN {X 0,Y 298.027,Z 720.362,A -85,B 0,C 180,E1 4135.381,E2 4135.381} C_VEL
LIN {X 0,Y 306.147,Z 658.891,A -85,B 0,C 180,E1 4134.517,E2 4134.517} C_VEL
LIN {X 0,Y 304.931,Z 655.945,A -85,B 0,C 180,E1 4131.134,E2 4131.134} C_VEL
LIN {X 0,Y 304.089,Z 654.869,A -85,B 0,C 180,E1 4125.528,E2 4125.528} C_VEL
LIN {X 0,Y 305.088,Z 656.049,A -85,B 0,C 180,E1 4119.671,E2 4119.671} C_VEL
LIN {X 0,Y 306.01,Z 658.752,A -85,B 0,C 180,E1 4116.995,E2 4116.995} C_VEL
LIN {X 0,Y 296.88,Z 726.204,A -85,B 0,C 180,E1 4116.098,E2 4116.098} C_VEL
LIN {X 0,Y 291.849,Z 749.773,A -85,B 0,C 180,E1 4115.756,E2 4115.756} C_VEL
LIN {X 0,Y 285.236,Z 773.12,A -85,B 0,C 180,E1 4115.316,E2 4115.316} C_VEL
LIN {X 0,Y 277.838,Z 793.781,A -85,B 0,C 180,E1 4114.814,E2 4114.814} C_VEL
LIN {X 0,Y 267.843,Z 816.753,A -85,B 0,C 180,E1 4114.093,E2 4114.093} C_VEL
LIN {X 0,Y 256.935,Z 837.871,A -85,B 0,C 180,E1 4113.245,E2 4113.245} C_VEL
LIN {X 0,Y 244.588,Z 857.987,A -85,B 0,C 180,E1 4112.211,E2 4112.211} C_VEL
LIN {X 0,Y 230.533,Z 877.868,A -85,B 0,C 180,E1 4110.9,E2 4110.9} C_VEL
LIN {X 0,Y 216.538,Z 895.096,A -85,B 0,C 180,E1 4109.427,E2 4109.427} C_VEL
LIN {X 0,Y 201.288,Z 911.554,A -85,B 0,C 180,E1 4107.593,E2 4107.593} C_VEL
LIN {X 0,Y 185.783,Z 926.419,A -85,B 0,C 180,E1 4105.409,E2 4105.409} C_VEL
LIN {X 0,Y 168.759,Z 940.725,A -85,B 0,C 180,E1 4102.533,E2 4102.533} C_VEL
LIN {X 0,Y 151.305,Z 953.778,A -85,B 0,C 180,E1 4098.86,E2 4098.86} C_VEL
LIN {X 0,Y 134.489,Z 964.786,A -85,B 0,C 180,E1 4094.314,E2 4094.314} C_VEL
LIN {X 0,Y 116.305,Z 975.4,A -85,B 0,C 180,E1 4087.596,E2 4087.596} C_VEL
LIN {X 0,Y 101.279,Z 983.353,A -85,B 0,C 180,E1 4079.558,E2 4079.558} C_VEL
LIN {X 0,Y 87.931,Z 989.896,A -85,B 0,C 180,E1 4068.544,E2 4068.544} C_VEL
LIN {X 0,Y 78.248,Z 994.868,A -85,B 0,C 180,E1 4054.627,E2 4054.627} C_VEL
LIN {X 0,Y 73.247,Z 997.991,A -85,B 0,C 180,E1 4038.959,E2 4038.959} C_VEL
LIN {X 0,Y 72.158,Z 999.436,A -85,B 0,C 180,E1 4027.146,E2 4027.146} C_VEL
LIN {X 0,Y 72.18,Z 1000.165,A -85,B 0,C 180,E1 4017.273,E2 4017.273} C_VEL
LIN {X 0,Y 73.598,Z 1000.463,A -85,B 0,C 180,E1 4003.861,E2 4003.861} C_VEL
LIN {X 0,Y 78.942,Z 999.832,A -85,B 0,C 180,E1 3988.774,E2 3988.774} C_VEL
LIN {X 0,Y 91.366,Z 997.425,A -85,B 0,C 180,E1 3973.029,E2 3973.029} C_VEL
LIN {X 0,Y 108.163,Z 993.445,A -85,B 0,C 180,E1 3961.591,E2 3961.591} C_VEL
LIN {X 0,Y 128.065,Z 987.557,A -85,B 0,C 180,E1 3953.276,E2 3953.276} C_VEL
LIN {X 0,Y 150.265,Z 979.817,A -85,B 0,C 180,E1 3947.126,E2 3947.126} C_VEL
LIN {X 0,Y 127.881,Z 988.53,A -85,B 0,C 180,E1 3941.13,E2 3941.13} C_VEL
LIN {X 0,Y 108.174,Z 995.266,A -85,B 0,C 180,E1 3933.072,E2 3933.072} C_VEL
LIN {X 0,Y 90.844,Z 1000.378,A -85,B 0,C 180,E1 3921.421,E2 3921.421} C_VEL
LIN {X 0,Y 78.942,Z 1003.7,A -85,B 0,C 180,E1 3906.559,E2 3906.559} C_VEL
LIN {X 0,Y 73.131,Z 1005.197,A -85,B 0,C 180,E1 3890.011,E2 3890.011} C_VEL
LIN {X 0,Y 72.064,Z 1005.439,A -85,B 0,C 180,E1 3877.197,E2 3877.197} C_VEL
LIN {X 0,Y 72.126,Z 1005.145,A -85,B 0,C 180,E1 3868.435,E2 3868.435} C_VEL
LIN {X 0,Y 72.219,Z 1004.211,A -85,B 0,C 180,E1 3858.039,E2 3858.039} C_VEL
LIN {X 0,Y 74.248,Z 1002.123,A -85,B 0,C 180,E1 3845.074,E2 3845.074} C_VEL
LIN {X 0,Y 75.148,Z 1000.874,A -85,B 0,C 180,E1 3839.249,E2 3839.249} C_VEL
LIN {X 0,Y 77.435,Z 996.547,A -85,B 0,C 180,E1 3823.191,E2 3823.191} C_VEL
LIN {X 0,Y 80.054,Z 995.008,A -85,B 0,C 180,E1 3819.296,E2 3819.296} C_VEL
LIN {X 0,Y 94.254,Z 988.372,A -85,B 0,C 180,E1 3807.821,E2 3807.821} C_VEL
LIN {X 0,Y 109.561,Z 980.58,A -85,B 0,C 180,E1 3800.004,E2 3800.004} C_VEL
LIN {X 0,Y 127.582,Z 970.487,A -85,B 0,C 180,E1 3793.71,E2 3793.71} C_VEL
LIN {X 0,Y 144.866,Z 959.508,A -85,B 0,C 180,E1 3789.345,E2 3789.345} C_VEL
LIN {X 0,Y 163.757,Z 945.882,A -85,B 0,C 180,E1 3785.726,E2 3785.726} C_VEL
LIN {X 0,Y 181.202,Z 931.616,A -85,B 0,C 180,E1 3783.099,E2 3783.099} C_VEL
LIN {X 0,Y 197.966,Z 915.827,A -85,B 0,C 180,E1 3781.036,E2 3781.036} C_VEL
LIN {X 0,Y 214.445,Z 898.246,A -85,B 0,C 180,E1 3779.343,E2 3779.343} C_VEL
LIN {X 0,Y 228.553,Z 881.042,A -85,B 0,C 180,E1 3778.104,E2 3778.104} C_VEL
LIN {X 0,Y 242.873,Z 860.967,A -85,B 0,C 180,E1 3777.005,E2 3777.005} C_VEL
LIN {X 0,Y 255.498,Z 840.574,A -85,B 0,C 180,E1 3776.156,E2 3776.156} C_VEL
LIN {X 0,Y 266.253,Z 820.001,A -85,B 0,C 180,E1 3775.508,E2 3775.508} C_VEL
LIN {X 0,Y 276.492,Z 796.749,A -85,B 0,C 180,E1 3774.952,E2 3774.952} C_VEL
LIN {X 0,Y 284.189,Z 775.49,A -85,B 0,C 180,E1 3774.58,E2 3774.58} C_VEL
LIN {X 0,Y 290.872,Z 751.978,A -85,B 0,C 180,E1 3774.262,E2 3774.262} C_VEL
LIN {X 0,Y 295.878,Z 728.39,A -85,B 0,C 180,E1 3773.954,E2 3773.954} C_VEL
LIN {X 0,Y 304.42,Z 665.669,A -85,B 0,C 180,E1 3773.114,E2 3773.114} C_VEL
LIN {X 0,Y 303.822,Z 663.869,A -85,B 0,C 180,E1 3771.101,E2 3771.101} C_VEL
LIN {X 0,Y 302.993,Z 662.794,A -85,B 0,C 180,E1 3765.475,E2 3765.475} C_VEL
LIN {X 0,Y 303.951,Z 663.956,A -85,B 0,C 180,E1 3759.793,E2 3759.793} C_VEL
LIN {X 0,Y 304.323,Z 665.52,A -85,B 0,C 180,E1 3758.406,E2 3758.406} C_VEL
LIN {X 0,Y 295.916,Z 726.795,A -85,B 0,C 180,E1 3757.63,E2 3757.63} C_VEL
LIN {X 0,Y 290.8,Z 750.447,A -85,B 0,C 180,E1 3757.311,E2 3757.311} C_VEL
LIN {X 0,Y 283.948,Z 774.251,A -85,B 0,C 180,E1 3756.895,E2 3756.895} C_VEL
LIN {X 0,Y 276.485,Z 794.821,A -85,B 0,C 180,E1 3756.433,E2 3756.433} C_VEL
LIN {X 0,Y 266.685,Z 817.034,A -85,B 0,C 180,E1 3755.791,E2 3755.791} C_VEL
LIN {X 0,Y 255.611,Z 838.243,A -85,B 0,C 180,E1 3755.009,E2 3755.009} C_VEL
LIN {X 0,Y 243.056,Z 858.452,A -85,B 0,C 180,E1 3754.055,E2 3754.055} C_VEL
LIN {X 0,Y 228.182,Z 879.139,A -85,B 0,C 180,E1 3752.791,E2 3752.791} C_VEL
LIN {X 0,Y 213.531,Z 896.867,A -85,B 0,C 180,E1 3751.377,E2 3751.377} C_VEL
LIN {X 0,Y 197.875,Z 913.288,A -85,B 0,C 180,E1 3749.648,E2 3749.648} C_VEL
LIN {X 0,Y 181.355,Z 928.666,A -85,B 0,C 180,E1 3747.493,E2 3747.493} C_VEL
LIN {X 0,Y 164.901,Z 942.01,A -85,B 0,C 180,E1 3744.919,E2 3744.919} C_VEL
LIN {X 0,Y 146.125,Z 955.464,A -85,B 0,C 180,E1 3741.243,E2 3741.243} C_VEL
LIN {X 0,Y 129.681,Z 965.828,A -85,B 0,C 180,E1 3737.071,E2 3737.071} C_VEL
LIN {X 0,Y 111.573,Z 975.895,A -85,B 0,C 180,E1 3730.835,E2 3730.835} C_VEL
LIN {X 0,Y 95.698,Z 983.836,A -85,B 0,C 180,E1 3722.885,E2 3722.885} C_VEL
LIN {X 0,Y 81.351,Z 990.337,A -85,B 0,C 180,E1 3711.613,E2 3711.613} C_VEL
LIN {X 0,Y 71.002,Z 995.147,A -85,B 0,C 180,E1 3697.256,E2 3697.256} C_VEL
LIN {X 0,Y 65.401,Z 998.239,A -85,B 0,C 180,E1 3680.292,E2 3680.292} C_VEL
LIN {X 0,Y 64.156,Z 999.708,A -85,B 0,C 180,E1 3667.041,E2 3667.041} C_VEL
LIN {X 0,Y 64.189,Z 1000.427,A -85,B 0,C 180,E1 3656.932,E2 3656.932} C_VEL
LIN {X 0,Y 65.906,Z 1000.804,A -85,B 0,C 180,E1 3641.881,E2 3641.881} C_VEL
LIN {X 0,Y 72.111,Z 1000.262,A -85,B 0,C 180,E1 3625.46,E2 3625.46} C_VEL
LIN {X 0,Y 86.078,Z 998.027,A -85,B 0,C 180,E1 3609.015,E2 3609.015} C_VEL
LIN {X 0,Y 103.058,Z 994.415,A -85,B 0,C 180,E1 3598.287,E2 3598.287} C_VEL
LIN {X 0,Y 123.856,Z 988.89,A -85,B 0,C 180,E1 3590.242,E2 3590.242} C_VEL
LIN {X 0,Y 134.741,Z 985.579,A -85,B 0,C 180,E1 3587.202,E2 3587.202} C_VEL
LIN {X 0,Y 112.511,Z 992.954,A -85,B 0,C 180,E1 3580.43,E2 3580.43} C_VEL
LIN {X 0,Y 92.844,Z 998.626,A -85,B 0,C 180,E1 3570.763,E2 3570.763} C_VEL
LIN {X 0,Y 76.877,Z 1002.456,A -85,B 0,C 180,E1 3556.777,E2 3556.777} C_VEL
LIN {X 0,Y 67.034,Z 1004.657,A -85,B 0,C 180,E1 3538.362,E2 3538.362} C_VEL
LIN {X 0,Y 64.148,Z 1005.133,A -85,B 0,C 180,E1 3520.807,E2 3520.807} C_VEL
LIN {X 0,Y 64.15,Z 1004.881,A -85,B 0,C 180,E1 3510.027,E2 3510.027} C_VEL
LIN {X 0,Y 64.179,Z 1004.064,A -85,B 0,C 180,E1 3498.942,E2 3498.942} C_VEL
LIN {X 0,Y 67.066,Z 1001.493,A -85,B 0,C 180,E1 3481.536,E2 3481.536} C_VEL
LIN {X 0,Y 74.184,Z 997.783,A -85,B 0,C 180,E1 3466.611,E2 3466.611} C_VEL
LIN {X 0,Y 80.054,Z 995.008,A -85,B 0,C 180,E1 3459.296,E2 3459.296} C_VEL
LIN {X 0,Y 83.625,Z 993.057,A -85,B 0,C 180,E1 3454.682,E2 3454.682} C_VEL
LIN {X 0,Y 92.505,Z 986.893,A -85,B 0,C 180,E1 3442.72,E2 3442.72} C_VEL
LIN {X 0,Y 96.85,Z 984.649,A -85,B 0,C 180,E1 3439.957,E2 3439.957} C_VEL
LIN {X 0,Y 114.916,Z 975.503,A -85,B 0,C 180,E1 3433.047,E2 3433.047} C_VEL
LIN {X 0,Y 133.3,Z 964.99,A -85,B 0,C 180,E1 3428.175,E2 3428.175} C_VEL
LIN {X 0,Y 151.884,Z 952.68,A -85,B 0,C 180,E1 3424.529,E2 3424.529} C_VEL
LIN {X 0,Y 170.021,Z 939.086,A -85,B 0,C 180,E1 3421.786,E2 3421.786} C_VEL
LIN {X 0,Y 187.273,Z 924.254,A -85,B 0,C 180,E1 3419.693,E2 3419.693} C_VEL
LIN {X 0,Y 204.562,Z 907.278,A -85,B 0,C 180,E1 3417.965,E2 3417.965} C_VEL
LIN {X 0,Y 219.693,Z 890.358,A -85,B 0,C 180,E1 3416.686,E2 3416.686} C_VEL
LIN {X 0,Y 234.218,Z 871.573,A -85,B 0,C 180,E1 3415.624,E2 3415.624} C_VEL
LIN {X 0,Y 247.452,Z 852.024,A -85,B 0,C 180,E1 3414.779,E2 3414.779} C_VEL
LIN {X 0,Y 258.779,Z 832.493,A -85,B 0,C 180,E1 3414.131,E2 3414.131} C_VEL
LIN {X 0,Y 270.129,Z 809.464,A -85,B 0,C 180,E1 3413.553,E2 3413.553} C_VEL
LIN {X 0,Y 279.427,Z 786.762,A -85,B 0,C 180,E1 3413.127,E2 3413.127} C_VEL
LIN {X 0,Y 286.902,Z 763.673,A -85,B 0,C 180,E1 3412.823,E2 3412.823} C_VEL
LIN {X 0,Y 293.129,Z 738.486,A -85,B 0,C 180,E1 3412.532,E2 3412.532} C_VEL
LIN {X 0,Y 297.234,Z 714.777,A -85,B 0,C 180,E1 3412.239,E2 3412.239} C_VEL
LIN {X 0,Y 302.894,Z 672.336,A -85,B 0,C 180,E1 3411.696,E2 3411.696} C_VEL
LIN {X 0,Y 302.38,Z 671.471,A -85,B 0,C 180,E1 3409.906,E2 3409.906} C_VEL
LIN {X 0,Y 301.898,Z 670.747,A -85,B 0,C 180,E1 3405.028,E2 3405.028} C_VEL
LIN {X 0,Y 302.827,Z 671.968,A -85,B 0,C 180,E1 3399.841,E2 3399.841} C_VEL
LIN {X 0,Y 295.113,Z 727.225,A -85,B 0,C 180,E1 3399.171,E2 3399.171} C_VEL
LIN {X 0,Y 289.931,Z 750.916,A -85,B 0,C 180,E1 3398.878,E2 3398.878} C_VEL
LIN {X 0,Y 282.871,Z 775.106,A -85,B 0,C 180,E1 3398.491,E2 3398.491} C_VEL
LIN {X 0,Y 274.866,Z 796.854,A -85,B 0,C 180,E1 3398.04,E2 3398.04} C_VEL
LIN {X 0,Y 265.166,Z 818.359,A -85,B 0,C 180,E1 3397.468,E2 3397.468} C_VEL
LIN {X 0,Y 254.041,Z 839.334,A -85,B 0,C 180,E1 3396.76,E2 3396.76} C_VEL
LIN {X 0,Y 241.48,Z 859.318,A -85,B 0,C 180,E1 3395.899,E2 3395.899} C_VEL
LIN {X 0,Y 226.564,Z 879.788,A -85,B 0,C 180,E1 3394.759,E2 3394.759} C_VEL
LIN {X 0,Y 211.727,Z 897.492,A -85,B 0,C 180,E1 3393.472,E2 3393.472} C_VEL
LIN {X 0,Y 196.021,Z 913.688,A -85,B 0,C 180,E1 3391.914,E2 3391.914} C_VEL
LIN {X 0,Y 179.045,Z 929.194,A -85,B 0,C 180,E1 3389.926,E2 3389.926} C_VEL
LIN {X 0,Y 161.981,Z 942.758,A -85,B 0,C 180,E1 3387.517,E2 3387.517} C_VEL
LIN {X 0,Y 143.026,Z 955.978,A -85,B 0,C 180,E1 3384.163,E2 3384.163} C_VEL
LIN {X 0,Y 125.196,Z 966.857,A -85,B 0,C 180,E1 3380.033,E2 3380.033} C_VEL
LIN {X 0,Y 107.227,Z 976.365,A -85,B 0,C 180,E1 3374.35,E2 3374.35} C_VEL
LIN {X 0,Y 90.478,Z 984.289,A -85,B 0,C 180,E1 3366.612,E2 3366.612} C_VEL
LIN {X 0,Y 75.043,Z 990.748,A -85,B 0,C 180,E1 3355.21,E2 3355.21} C_VEL
LIN {X 0,Y 63.647,Z 995.53,A -85,B 0,C 180,E1 3339.923,E2 3339.923} C_VEL
LIN {X 0,Y 57.416,Z 998.597,A -85,B 0,C 180,E1 3320.953,E2 3320.953} C_VEL
LIN {X 0,Y 56.154,Z 999.97,A -85,B 0,C 180,E1 3306.905,E2 3306.905} C_VEL
LIN {X 0,Y 56.257,Z 1000.738,A -85,B 0,C 180,E1 3294.849,E2 3294.849} C_VEL
LIN {X 0,Y 58.908,Z 1001.129,A -85,B 0,C 180,E1 3277.038,E2 3277.038} C_VEL
LIN {X 0,Y 67.082,Z 1000.553,A -85,B 0,C 180,E1 3259.146,E2 3259.146} C_VEL
LIN {X 0,Y 83.689,Z 998.199,A -85,B 0,C 180,E1 3242.742,E2 3242.742} C_VEL
LIN {X 0,Y 102.842,Z 994.466,A -85,B 0,C 180,E1 3232.741,E2 3232.741} C_VEL
LIN {X 0,Y 118.948,Z 990.555,A -85,B 0,C 180,E1 3227.238,E2 3227.238} C_VEL
LIN {X 0,Y 97.051,Z 996.595,A -85,B 0,C 180,E1 3219.498,E2 3219.498} C_VEL
LIN {X 0,Y 77.955,Z 1001.067,A -85,B 0,C 180,E1 3207.874,E2 3207.874} C_VEL
LIN {X 0,Y 63.934,Z 1003.69,A -85,B 0,C 180,E1 3191.093,E2 3191.093} C_VEL
LIN {X 0,Y 56.897,Z 1004.845,A -85,B 0,C 180,E1 3169.537,E2 3169.537} C_VEL
LIN {X 0,Y 56.1,Z 1004.689,A -85,B 0,C 180,E1 3153.62,E2 3153.62} C_VEL
LIN {X 0,Y 56.105,Z 1004.107,A -85,B 0,C 180,E1 3143.893,E2 3143.893} C_VEL
LIN {X 0,Y 57.442,Z 1002.454,A -85,B 0,C 180,E1 3127.29,E2 3127.29} C_VEL
LIN {X 0,Y 64.776,Z 998.709,A -85,B 0,C 180,E1 3107.26,E2 3107.26} C_VEL
LIN {X 0,Y 76.364,Z 993.782,A -85,B 0,C 180,E1 3093.118,E2 3093.118} C_VEL
LIN {X 0,Y 92.704,Z 986.562,A -85,B 0,C 180,E1 3081.999,E2 3081.999} C_VEL
LIN {X 0,Y 96.85,Z 984.649,A -85,B 0,C 180,E1 3079.957,E2 3079.957} C_VEL
LIN {X 0,Y 102.022,Z 981.965,A -85,B 0,C 180,E1 3076.999,E2 3076.999} C_VEL
LIN {X 0,Y 114.628,Z 974.015,A -85,B 0,C 180,E1 3068.959,E2 3068.959} C_VEL
LIN {X 0,Y 119.59,Z 971.164,A -85,B 0,C 180,E1 3067.284,E2 3067.284} C_VEL
LIN {X 0,Y 138.196,Z 960.12,A -85,B 0,C 180,E1 3063.458,E2 3063.458} C_VEL
LIN {X 0,Y 156.949,Z 947.456,A -85,B 0,C 180,E1 3060.557,E2 3060.557} C_VEL
LIN {X 0,Y 174,Z 934.202,A -85,B 0,C 180,E1 3058.471,E2 3058.471} C_VEL
LIN {X 0,Y 192.772,Z 917.524,A -85,B 0,C 180,E1 3056.612,E2 3056.612} C_VEL
LIN {X 0,Y 209.143,Z 900.898,A -85,B 0,C 180,E1 3055.274,E2 3055.274} C_VEL
LIN {X 0,Y 224.587,Z 882.709,A -85,B 0,C 180,E1 3054.198,E2 3054.198} C_VEL
LIN {X 0,Y 238.824,Z 863.563,A -85,B 0,C 180,E1 3053.341,E2 3053.341} C_VEL
LIN {X 0,Y 251.282,Z 844.127,A -85,B 0,C 180,E1 3052.684,E2 3052.684} C_VEL
LIN {X 0,Y 263.015,Z 822.701,A -85,B 0,C 180,E1 3052.133,E2 3052.133} C_VEL
LIN {X 0,Y 272.76,Z 801.733,A -85,B 0,C 180,E1 3051.726,E2 3051.726} C_VEL
LIN {X 0,Y 281.125,Z 779.705,A -85,B 0,C 180,E1 3051.408,E2 3051.408} C_VEL
LIN {X 0,Y 288.239,Z 756.554,A -85,B 0,C 180,E1 3051.16,E2 3051.16} C_VEL
LIN {X 0,Y 293.439,Z 733.787,A -85,B 0,C 180,E1 3050.918,E2 3050.918} C_VEL
LIN {X 0,Y 298.319,Z 702.259,A -85,B 0,C 180,E1 3050.554,E2 3050.554} C_VEL
LIN {X 0,Y 301.372,Z 679.494,A -85,B 0,C 180,E1 3050.258,E2 3050.258} C_VEL
LIN {X 0,Y 300.803,Z 678.657,A -85,B 0,C 180,E1 3045.17,E2 3045.17} C_VEL
LIN {X 0,Y 301.288,Z 679.596,A -85,B 0,C 180,E1 3041.261,E2 3041.261} C_VEL
LIN {X 0,Y 294.409,Z 728,A -85,B 0,C 180,E1 3040.715,E2 3040.715} C_VEL
LIN {X 0,Y 289.216,Z 751.496,A -85,B 0,C 180,E1 3040.451,E2 3040.451} C_VEL
LIN {X 0,Y 282.21,Z 775.332,A -85,B 0,C 180,E1 3040.108,E2 3040.108} C_VEL
LIN {X 0,Y 274.436,Z 796.381,A -85,B 0,C 180,E1 3039.719,E2 3039.719} C_VEL
LIN {X 0,Y 264.663,Z 818.047,A -85,B 0,C 180,E1 3039.207,E2 3039.207} C_VEL
LIN {X 0,Y 253.442,Z 839.132,A -85,B 0,C 180,E1 3038.574,E2 3038.574} C_VEL
LIN {X 0,Y 240.766,Z 859.162,A -85,B 0,C 180,E1 3037.807,E2 3037.807} C_VEL
LIN {X 0,Y 226.025,Z 879.298,A -85,B 0,C 180,E1 3036.814,E2 3036.814} C_VEL
LIN {X 0,Y 211.371,Z 896.694,A -85,B 0,C 180,E1 3035.697,E2 3035.697} C_VEL
LIN {X 0,Y 195.259,Z 913.286,A -85,B 0,C 180,E1 3034.296,E2 3034.296} C_VEL
LIN {X 0,Y 178.019,Z 928.933,A -85,B 0,C 180,E1 3032.525,E2 3032.525} C_VEL
LIN {X 0,Y 160.924,Z 942.352,A -85,B 0,C 180,E1 3030.416,E2 3030.416} C_VEL
LIN {X 0,Y 142.175,Z 955.295,A -85,B 0,C 180,E1 3027.529,E2 3027.529} C_VEL
LIN {X 0,Y 123.777,Z 966.278,A -85,B 0,C 180,E1 3023.854,E2 3023.854} C_VEL
LIN {X 0,Y 104.185,Z 976.391,A -85,B 0,C 180,E1 3018.438,E2 3018.438} C_VEL
LIN {X 0,Y 86.115,Z 984.528,A -85,B 0,C 180,E1 3010.997,E2 3010.997} C_VEL
LIN {X 0,Y 69.779,Z 990.889,A -85,B 0,C 180,E1 3000.07,E2 3000.07} C_VEL
LIN {X 0,Y 56.538,Z 995.874,A -85,B 0,C 180,E1 2983.413,E2 2983.413} C_VEL
LIN {X 0,Y 49.643,Z 998.828,A -85,B 0,C 180,E1 2963.024,E2 2963.024} C_VEL
LIN {X 0,Y 48.149,Z 1000.231,A -85,B 0,C 180,E1 2946.724,E2 2946.724} C_VEL
LIN {X 0,Y 48.333,Z 1001.021,A -85,B 0,C 180,E1 2933.092,E2 2933.092} C_VEL
LIN {X 0,Y 51.992,Z 1001.465,A -85,B 0,C 180,E1 2912.143,E2 2912.143} C_VEL
LIN {X 0,Y 62.49,Z 1000.891,A -85,B 0,C 180,E1 2892.457,E2 2892.457} C_VEL
LIN {X 0,Y 81.819,Z 998.48,A -85,B 0,C 180,E1 2876.5,E2 2876.5} C_VEL
LIN {X 0,Y 103.16,Z 994.635,A -85,B 0,C 180,E1 2867.303,E2 2867.303} C_VEL
LIN {X 0,Y 80.965,Z 999.572,A -85,B 0,C 180,E1 2857.9,E2 2857.9} C_VEL
LIN {X 0,Y 61.4,Z 1002.992,A -85,B 0,C 180,E1 2841.455,E2 2841.455} C_VEL
LIN {X 0,Y 51.37,Z 1004.291,A -85,B 0,C 180,E1 2821.742,E2 2821.742} C_VEL
LIN {X 0,Y 48.125,Z 1004.426,A -85,B 0,C 180,E1 2799.604,E2 2799.604} C_VEL
LIN {X 0,Y 48.15,Z 1004.028,A -85,B 0,C 180,E1 2788.846,E2 2788.846} C_VEL
LIN {X 0,Y 48.426,Z 1003.063,A -85,B 0,C 180,E1 2774.468,E2 2774.468} C_VEL
LIN {X 0,Y 52.766,Z 1000.59,A -85,B 0,C 180,E1 2754.068,E2 2754.068} C_VEL
LIN {X 0,Y 63.775,Z 996.332,A -85,B 0,C 180,E1 2735.438,E2 2735.438} C_VEL
LIN {X 0,Y 79.087,Z 990.267,A -85,B 0,C 180,E1 2722.708,E2 2722.708} C_VEL
LIN {X 0,Y 96.881,Z 982.603,A -85,B 0,C 180,E1 2714.122,E2 2714.122} C_VEL
LIN {X 0,Y 115.18,Z 973.475,A -85,B 0,C 180,E1 2708.385,E2 2708.385} C_VEL
LIN {X 0,Y 119.59,Z 971.164,A -85,B 0,C 180,E1 2707.284,E2 2707.284} C_VEL
LIN {X 0,Y 125.372,Z 967.738,A -85,B 0,C 180,E1 2705.46,E2 2705.46} C_VEL
LIN {X 0,Y 139.535,Z 958.031,A -85,B 0,C 180,E1 2700.035,E2 2700.035} C_VEL
LIN {X 0,Y 144.605,Z 954.555,A -85,B 0,C 180,E1 2698.997,E2 2698.997} C_VEL
LIN {X 0,Y 163.197,Z 941.438,A -85,B 0,C 180,E1 2696.784,E2 2696.784} C_VEL
LIN {X 0,Y 181.616,Z 926.424,A -85,B 0,C 180,E1 2695.043,E2 2695.043} C_VEL
LIN {X 0,Y 198.67,Z 910.599,A -85,B 0,C 180,E1 2693.726,E2 2693.726} C_VEL
LIN {X 0,Y 214.681,Z 893.353,A -85,B 0,C 180,E1 2692.68,E2 2692.68} C_VEL
LIN {X 0,Y 230.867,Z 873.327,A -85,B 0,C 180,E1 2691.782,E2 2691.782} C_VEL
LIN {X 0,Y 243.824,Z 854.835,A -85,B 0,C 180,E1 2691.157,E2 2691.157} C_VEL
LIN {X 0,Y 255.829,Z 834.868,A -85,B 0,C 180,E1 2690.642,E2 2690.642} C_VEL
LIN {X 0,Y 266.794,Z 813.688,A -85,B 0,C 180,E1 2690.227,E2 2690.227} C_VEL
LIN {X 0,Y 276.195,Z 791.599,A -85,B 0,C 180,E1 2689.906,E2 2689.906} C_VEL
LIN {X 0,Y 284.735,Z 766.859,A -85,B 0,C 180,E1 2689.655,E2 2689.655} C_VEL
LIN {X 0,Y 290.958,Z 743.642,A -85,B 0,C 180,E1 2689.453,E2 2689.453} C_VEL
LIN {X 0,Y 295.409,Z 719.845,A -85,B 0,C 180,E1 2689.207,E2 2689.207} C_VEL
LIN {X 0,Y 299.989,Z 687.102,A -85,B 0,C 180,E1 2688.853,E2 2688.853} C_VEL
LIN {X 0,Y 299.721,Z 686.67,A -85,B 0,C 180,E1 2684.57,E2 2684.57} C_VEL
LIN {X 0,Y 299.904,Z 687.215,A -85,B 0,C 180,E1 2682.702,E2 2682.702} C_VEL
LIN {X 0,Y 293.853,Z 728.749,A -85,B 0,C 180,E1 2682.265,E2 2682.265} C_VEL
LIN {X 0,Y 288.656,Z 752.031,A -85,B 0,C 180,E1 2682.031,E2 2682.031} C_VEL
LIN {X 0,Y 281.376,Z 776.451,A -85,B 0,C 180,E1 2681.716,E2 2681.716} C_VEL
LIN {X 0,Y 273.259,Z 798.134,A -85,B 0,C 180,E1 2681.358,E2 2681.358} C_VEL
LIN {X 0,Y 263.415,Z 819.52,A -85,B 0,C 180,E1 2680.907,E2 2680.907} C_VEL
LIN {X 0,Y 252.111,Z 840.415,A -85,B 0,C 180,E1 2680.348,E2 2680.348} C_VEL
LIN {X 0,Y 239.828,Z 859.66,A -85,B 0,C 180,E1 2679.698,E2 2679.698} C_VEL
LIN {X 0,Y 224.627,Z 880.203,A -85,B 0,C 180,E1 2678.805,E2 2678.805} C_VEL
LIN {X 0,Y 209.47,Z 897.979,A -85,B 0,C 180,E1 2677.795,E2 2677.795} C_VEL
LIN {X 0,Y 192.89,Z 914.682,A -85,B 0,C 180,E1 2676.534,E2 2676.534} C_VEL
LIN {X 0,Y 175.425,Z 930.147,A -85,B 0,C 180,E1 2674.963,E2 2674.963} C_VEL
LIN {X 0,Y 158.067,Z 943.491,A -85,B 0,C 180,E1 2673.084,E2 2673.084} C_VEL
LIN {X 0,Y 138.008,Z 956.883,A -85,B 0,C 180,E1 2670.359,E2 2670.359} C_VEL
LIN {X 0,Y 119.19,Z 967.754,A -85,B 0,C 180,E1 2666.991,E2 2666.991} C_VEL
LIN {X 0,Y 99.892,Z 977.223,A -85,B 0,C 180,E1 2662.224,E2 2662.224} C_VEL
LIN {X 0,Y 80.762,Z 985.353,A -85,B 0,C 180,E1 2655.112,E2 2655.112} C_VEL
LIN {X 0,Y 63.572,Z 991.533,A -85,B 0,C 180,E1 2644.452,E2 2644.452} C_VEL
LIN {X 0,Y 48.979,Z 996.419,A -85,B 0,C 180,E1 2626.569,E2 2626.569} C_VEL
LIN {X 0,Y 41.706,Z 999.171,A -85,B 0,C 180,E1 2604.455,E2 2604.455} C_VEL
LIN {X 0,Y 40.145,Z 1000.486,A -85,B 0,C 180,E1 2586.47,E2 2586.47} C_VEL
LIN {X 0,Y 40.519,Z 1001.32,A -85,B 0,C 180,E1 2569.912,E2 2569.912} C_VEL
LIN {X 0,Y 46.153,Z 1001.796,A -85,B 0,C 180,E1 2544.312,E2 2544.312} C_VEL
LIN {X 0,Y 59.2,Z 1001.216,A -85,B 0,C 180,E1 2524.474,E2 2524.474} C_VEL
LIN {X 0,Y 80.135,Z 998.901,A -85,B 0,C 180,E1 2510.414,E2 2510.414} C_VEL
LIN {X 0,Y 87.133,Z 997.895,A -85,B 0,C 180,E1 2507.341,E2 2507.341} C_VEL
LIN {X 0,Y 66.427,Z 1001.468,A -85,B 0,C 180,E1 2496.721,E2 2496.721} C_VEL
LIN {X 0,Y 48.442,Z 1003.703,A -85,B 0,C 180,E1 2476.304,E2 2476.304} C_VEL
LIN {X 0,Y 40.972,Z 1004.135,A -85,B 0,C 180,E1 2451.517,E2 2451.517} C_VEL
LIN {X 0,Y 40.127,Z 1003.801,A -85,B 0,C 180,E1 2432.9,E2 2432.9} C_VEL
LIN {X 0,Y 40.157,Z 1003.239,A -85,B 0,C 180,E1 2420.007,E2 2420.007} C_VEL
LIN {X 0,Y 44.165,Z 1000.872,A -85,B 0,C 180,E1 2393.992,E2 2393.992} C_VEL
LIN {X 0,Y 54.425,Z 997.244,A -85,B 0,C 180,E1 2374.299,E2 2374.299} C_VEL
LIN {X 0,Y 71.29,Z 991.359,A -85,B 0,C 180,E1 2359.667,E2 2359.667} C_VEL
LIN {X 0,Y 88.708,Z 984.444,A -85,B 0,C 180,E1 2351.412,E2 2351.412} C_VEL
LIN {X 0,Y 109.413,Z 974.853,A -85,B 0,C 180,E1 2345.275,E2 2345.275} C_VEL
LIN {X 0,Y 129.141,Z 964.224,A -85,B 0,C 180,E1 2341.329,E2 2341.329} C_VEL
LIN {X 0,Y 144.605,Z 954.555,A -85,B 0,C 180,E1 2338.997,E2 2338.997} C_VEL
LIN {X 0,Y 150.456,Z 950.476,A -85,B 0,C 180,E1 2337.839,E2 2337.839} C_VEL
LIN {X 0,Y 164.963,Z 939.128,A -85,B 0,C 180,E1 2333.996,E2 2333.996} C_VEL
LIN {X 0,Y 169.932,Z 935.079,A -85,B 0,C 180,E1 2333.321,E2 2333.321} C_VEL
LIN {X 0,Y 187.746,Z 919.98,A -85,B 0,C 180,E1 2332.037,E2 2332.037} C_VEL
LIN {X 0,Y 204.429,Z 903.604,A -85,B 0,C 180,E1 2331.038,E2 2331.038} C_VEL
LIN {X 0,Y 221.162,Z 884.743,A -85,B 0,C 180,E1 2330.193,E2 2330.193} C_VEL
LIN {X 0,Y 235.831,Z 865.703,A -85,B 0,C 180,E1 2329.561,E2 2329.561} C_VEL
LIN {X 0,Y 248.942,Z 845.718,A -85,B 0,C 180,E1 2329.068,E2 2329.068} C_VEL
LIN {X 0,Y 261.008,Z 824.337,A -85,B 0,C 180,E1 2328.672,E2 2328.672} C_VEL
LIN {X 0,Y 270.449,Z 804.492,A -85,B 0,C 180,E1 2328.397,E2 2328.397} C_VEL
LIN {X 0,Y 279.621,Z 781.274,A -85,B 0,C 180,E1 2328.158,E2 2328.158} C_VEL
LIN {X 0,Y 286.95,Z 758.183,A -85,B 0,C 180,E1 2327.989,E2 2327.989} C_VEL
LIN {X 0,Y 292.461,Z 734.719,A -85,B 0,C 180,E1 2327.799,E2 2327.799} C_VEL
LIN {X 0,Y 297.063,Z 706.482,A -85,B 0,C 180,E1 2327.518,E2 2327.518} C_VEL
LIN {X 0,Y 298.677,Z 694.676,A -85,B 0,C 180,E1 2327.382,E2 2327.382} C_VEL
LIN {X 0,Y 298.645,Z 694.714,A -85,B 0,C 180,E1 2324.158,E2 2324.158} C_VEL
LIN {X 0,Y 293.328,Z 730.109,A -85,B 0,C 180,E1 2323.813,E2 2323.813} C_VEL
LIN {X 0,Y 288.158,Z 752.998,A -85,B 0,C 180,E1 2323.611,E2 2323.611} C_VEL
LIN {X 0,Y 280.962,Z 776.903,A -85,B 0,C 180,E1 2323.342,E2 2323.342} C_VEL
LIN {X 0,Y 272.798,Z 798.601,A -85,B 0,C 180,E1 2323.032,E2 2323.032} C_VEL
LIN {X 0,Y 262.896,Z 819.979,A -85,B 0,C 180,E1 2322.643,E2 2322.643} C_VEL
LIN {X 0,Y 251.518,Z 840.841,A -85,B 0,C 180,E1 2322.161,E2 2322.161} C_VEL
LIN {X 0,Y 239.15,Z 860.073,A -85,B 0,C 180,E1 2321.603,E2 2321.603} C_VEL
LIN {X 0,Y 223.833,Z 880.594,A -85,B 0,C 180,E1 2320.838,E2 2320.838} C_VEL
LIN {X 0,Y 208.545,Z 898.368,A -85,B 0,C 180,E1 2319.973,E2 2319.973} C_VEL
LIN {X 0,Y 191.803,Z 915.082,A -85,B 0,C 180,E1 2318.895,E2 2318.895} C_VEL
LIN {X 0,Y 174.136,Z 930.553,A -85,B 0,C 180,E1 2317.552,E2 2317.552} C_VEL
LIN {X 0,Y 156.538,Z 943.91,A -85,B 0,C 180,E1 2315.945,E2 2315.945} C_VEL
LIN {X 0,Y 136.134,Z 957.291,A -85,B 0,C 180,E1 2313.61,E2 2313.61} C_VEL
LIN {X 0,Y 116.893,Z 968.154,A -85,B 0,C 180,E1 2310.713,E2 2310.713} C_VEL
LIN {X 0,Y 97.006,Z 977.601,A -85,B 0,C 180,E1 2306.568,E2 2306.568} C_VEL
LIN {X 0,Y 77.69,Z 985.488,A -85,B 0,C 180,E1 2300.513,E2 2300.513} C_VEL
LIN {X 0,Y 58.632,Z 991.895,A -85,B 0,C 180,E1 2290.351,E2 2290.351} C_VEL
LIN {X 0,Y 42.333,Z 996.762,A -85,B 0,C 180,E1 2272.159,E2 2272.159} C_VEL
LIN {X 0,Y 33.804,Z 999.506,A -85,B 0,C 180,E1 2246.557,E2 2246.557} C_VEL
LIN {X 0,Y 32.116,Z 1000.817,A -85,B 0,C 180,E1 2224.101,E2 2224.101} C_VEL
LIN {X 0,Y 33.059,Z 1001.654,A -85,B 0,C 180,E1 2203.384,E2 2203.384} C_VEL
LIN {X 0,Y 41.651,Z 1002.129,A -85,B 0,C 180,E1 2173.896,E2 2173.896} C_VEL
LIN {X 0,Y 58.245,Z 1001.489,A -85,B 0,C 180,E1 2154.957,E2 2154.957} C_VEL
LIN {X 0,Y 71.137,Z 1000.322,A -85,B 0,C 180,E1 2147.49,E2 2147.49} C_VEL
LIN {X 0,Y 51.103,Z 1002.773,A -85,B 0,C 180,E1 2134.233,E2 2134.233} C_VEL
LIN {X 0,Y 35.961,Z 1003.823,A -85,B 0,C 180,E1 2107.77,E2 2107.77} C_VEL
LIN {X 0,Y 32.125,Z 1003.552,A -85,B 0,C 180,E1 2079.007,E2 2079.007} C_VEL
LIN {X 0,Y 32.136,Z 1003.156,A -85,B 0,C 180,E1 2066.487,E2 2066.487} C_VEL
LIN {X 0,Y 33.798,Z 1001.749,A -85,B 0,C 180,E1 2041.809,E2 2041.809} C_VEL
LIN {X 0,Y 44.409,Z 998.346,A -85,B 0,C 180,E1 2013.661,E2 2013.661} C_VEL
LIN {X 0,Y 59.971,Z 993.538,A -85,B 0,C 180,E1 1998.236,E2 1998.236} C_VEL
LIN {X 0,Y 79.827,Z 986.547,A -85,B 0,C 180,E1 1988.475,E2 1988.475} C_VEL
LIN {X 0,Y 99.221,Z 978.397,A -85,B 0,C 180,E1 1982.886,E2 1982.886} C_VEL
LIN {X 0,Y 119.969,Z 968.068,A -85,B 0,C 180,E1 1978.925,E2 1978.925} C_VEL
LIN {X 0,Y 139.269,Z 956.871,A -85,B 0,C 180,E1 1976.294,E2 1976.294} C_VEL
LIN {X 0,Y 158.734,Z 943.605,A -85,B 0,C 180,E1 1974.27,E2 1974.27} C_VEL
LIN {X 0,Y 169.932,Z 935.079,A -85,B 0,C 180,E1 1973.321,E2 1973.321} C_VEL
LIN {X 0,Y 175.625,Z 930.44,A -85,B 0,C 180,E1 1972.547,E2 1972.547} C_VEL
LIN {X 0,Y 188.972,Z 918.156,A -85,B 0,C 180,E1 1969.79,E2 1969.79} C_VEL
LIN {X 0,Y 194.446,Z 912.905,A -85,B 0,C 180,E1 1969.222,E2 1969.222} C_VEL
LIN {X 0,Y 211.71,Z 895.023,A -85,B 0,C 180,E1 1968.463,E2 1968.463} C_VEL
LIN {X 0,Y 226.976,Z 876.905,A -85,B 0,C 180,E1 1967.895,E2 1967.895} C_VEL
LIN {X 0,Y 241.203,Z 857.136,A -85,B 0,C 180,E1 1967.436,E2 1967.436} C_VEL
LIN {X 0,Y 254.583,Z 835.503,A -85,B 0,C 180,E1 1967.063,E2 1967.063} C_VEL
LIN {X 0,Y 265.436,Z 814.875,A -85,B 0,C 180,E1 1966.8,E2 1966.8} C_VEL
LIN {X 0,Y 275.142,Z 792.577,A -85,B 0,C 180,E1 1966.592,E2 1966.592} C_VEL
LIN {X 0,Y 283.405,Z 769.407,A -85,B 0,C 180,E1 1966.448,E2 1966.448} C_VEL
LIN {X 0,Y 289.566,Z 747.173,A -85,B 0,C 180,E1 1966.324,E2 1966.324} C_VEL
LIN {X 0,Y 294.594,Z 722.354,A -85,B 0,C 180,E1 1966.122,E2 1966.122} C_VEL
LIN {X 0,Y 297.534,Z 702.435,A -85,B 0,C 180,E1 1965.898,E2 1965.898} C_VEL
LIN {X 0,Y 297.511,Z 702.517,A -85,B 0,C 180,E1 1965.622,E2 1965.622} C_VEL
LIN {X 0,Y 292.538,Z 733.538,A -85,B 0,C 180,E1 1965.353,E2 1965.353} C_VEL
LIN {X 0,Y 287.009,Z 757.158,A -85,B 0,C 180,E1 1965.172,E2 1965.172} C_VEL
LIN {X 0,Y 279.776,Z 780,A -85,B 0,C 180,E1 1964.943,E2 1964.943} C_VEL
LIN {X 0,Y 270.578,Z 803.352,A -85,B 0,C 180,E1 1964.647,E2 1964.647} C_VEL
LIN {X 0,Y 261.125,Z 823.184,A -85,B 0,C 180,E1 1964.333,E2 1964.333} C_VEL
LIN {X 0,Y 249.185,Z 844.337,A -85,B 0,C 180,E1 1963.912,E2 1963.912} C_VEL
LIN {X 0,Y 236.253,Z 864.033,A -85,B 0,C 180,E1 1963.419,E2 1963.419} C_VEL
LIN {X 0,Y 221.83,Z 882.755,A -85,B 0,C 180,E1 1962.819,E2 1962.819} C_VEL
LIN {X 0,Y 205.935,Z 900.781,A -85,B 0,C 180,E1 1962.07,E2 1962.07} C_VEL
LIN {X 0,Y 190.052,Z 916.379,A -85,B 0,C 180,E1 1961.222,E2 1961.222} C_VEL
LIN {X 0,Y 171.226,Z 932.457,A -85,B 0,C 180,E1 1960.04,E2 1960.04} C_VEL
LIN {X 0,Y 152.445,Z 946.379,A -85,B 0,C 180,E1 1958.609,E2 1958.609} C_VEL
LIN {X 0,Y 132.74,Z 958.8,A -85,B 0,C 180,E1 1956.736,E2 1956.736} C_VEL
LIN {X 0,Y 112.18,Z 969.955,A -85,B 0,C 180,E1 1954.145,E2 1954.145} C_VEL
LIN {X 0,Y 92.782,Z 978.785,A -85,B 0,C 180,E1 1950.754,E2 1950.754} C_VEL
LIN {X 0,Y 70.902,Z 987.082,A -85,B 0,C 180,E1 1944.831,E2 1944.831} C_VEL
LIN {X 0,Y 51.774,Z 993.034,A -85,B 0,C 180,E1 1935.556,E2 1935.556} C_VEL
LIN {X 0,Y 34.1,Z 997.601,A -85,B 0,C 180,E1 1916.035,E2 1916.035} C_VEL
LIN {X 0,Y 25.336,Z 1000.087,A -85,B 0,C 180,E1 1885.404,E2 1885.404} C_VEL
LIN {X 0,Y 24.139,Z 1001.147,A -85,B 0,C 180,E1 1860.113,E2 1860.113} C_VEL
LIN {X 0,Y 27.228,Z 1002.082,A -85,B 0,C 180,E1 1828.068,E2 1828.068} C_VEL
LIN {X 0,Y 39.031,Z 1002.467,A -85,B 0,C 180,E1 1801.106,E2 1801.106} C_VEL
LIN {X 0,Y 54.743,Z 1001.976,A -85,B 0,C 180,E1 1787.6,E2 1787.6} C_VEL
LIN {X 0,Y 35.813,Z 1003.324,A -85,B 0,C 180,E1 1769.839,E2 1769.839} C_VEL
LIN {X 0,Y 24.681,Z 1003.332,A -85,B 0,C 180,E1 1731.316,E2 1731.316} C_VEL
LIN {X 0,Y 24.181,Z 1002.87,A -85,B 0,C 180,E1 1710.072,E2 1710.072} C_VEL
LIN {X 0,Y 25.156,Z 1001.84,A -85,B 0,C 180,E1 1684.152,E2 1684.152} C_VEL
LIN {X 0,Y 33.657,Z 999.397,A -85,B 0,C 180,E1 1653.812,E2 1653.812} C_VEL
LIN {X 0,Y 51.51,Z 994.689,A -85,B 0,C 180,E1 1634.089,E2 1634.089} C_VEL
LIN {X 0,Y 70.239,Z 988.781,A -85,B 0,C 180,E1 1625.135,E2 1625.135} C_VEL
LIN {X 0,Y 91.959,Z 980.455,A -85,B 0,C 180,E1 1619.364,E2 1619.364} C_VEL
LIN {X 0,Y 112.229,Z 971.129,A -85,B 0,C 180,E1 1615.951,E2 1615.951} C_VEL
LIN {X 0,Y 132.84,Z 959.787,A -85,B 0,C 180,E1 1613.516,E2 1613.516} C_VEL
LIN {X 0,Y 152.508,Z 947.24,A -85,B 0,C 180,E1 1611.782,E2 1611.782} C_VEL
LIN {X 0,Y 171.298,Z 933.205,A -85,B 0,C 180,E1 1610.48,E2 1610.48} C_VEL
LIN {X 0,Y 190.488,Z 916.627,A -85,B 0,C 180,E1 1609.413,E2 1609.413} C_VEL
LIN {X 0,Y 194.446,Z 912.905,A -85,B 0,C 180,E1 1609.222,E2 1609.222} C_VEL
LIN {X 0,Y 199.849,Z 907.635,A -85,B 0,C 180,E1 1608.69,E2 1608.69} C_VEL
LIN {X 0,Y 212.476,Z 893.99,A -85,B 0,C 180,E1 1606.537,E2 1606.537} C_VEL
LIN {X 0,Y 217.424,Z 888.211,A -85,B 0,C 180,E1 1606.121,E2 1606.121} C_VEL
LIN {X 0,Y 232.079,Z 869.73,A -85,B 0,C 180,E1 1605.741,E2 1605.741} C_VEL
LIN {X 0,Y 241.198,Z 856.83,A -85,B 0,C 180,E1 1605.517,E2 1605.517} C_VEL
LIN {X 0,Y 227.098,Z 876.296,A -85,B 0,C 180,E1 1605.068,E2 1605.068} C_VEL
LIN {X 0,Y 211.604,Z 894.552,A -85,B 0,C 180,E1 1604.525,E2 1604.525} C_VEL
LIN {X 0,Y 194.614,Z 912.007,A -85,B 0,C 180,E1 1603.852,E2 1603.852} C_VEL
LIN {X 0,Y 177.632,Z 927.127,A -85,B 0,C 180,E1 1603.076,E2 1603.076} C_VEL
LIN {X 0,Y 158.664,Z 941.757,A -85,B 0,C 180,E1 1602.051,E2 1602.051} C_VEL
LIN {X 0,Y 139.725,Z 954.434,A -85,B 0,C 180,E1 1600.791,E2 1600.791} C_VEL
LIN {X 0,Y 119.816,Z 965.727,A -85,B 0,C 180,E1 1599.123,E2 1599.123} C_VEL
LIN {X 0,Y 98.982,Z 975.823,A -85,B 0,C 180,E1 1596.764,E2 1596.764} C_VEL
LIN {X 0,Y 77.771,Z 984.22,A -85,B 0,C 180,E1 1593.255,E2 1593.255} C_VEL
LIN {X 0,Y 54.938,Z 991.521,A -85,B 0,C 180,E1 1586.783,E2 1586.783} C_VEL
LIN {X 0,Y 36.273,Z 996.252,A -85,B 0,C 180,E1 1575.71,E2 1575.71} C_VEL
LIN {X 0,Y 19.858,Z 999.78,A -85,B 0,C 180,E1 1544.49,E2 1544.49} C_VEL
LIN {X 0,Y 16.116,Z 1001.216,A -85,B 0,C 180,E1 1504.142,E2 1504.142} C_VEL
LIN {X 0,Y 18.86,Z 1002.146,A -85,B 0,C 180,E1 1465.108,E2 1465.108} C_VEL
LIN {X 0,Y 35.591,Z 1002.82,A -85,B 0,C 180,E1 1429.764,E2 1429.764} C_VEL
LIN {X 0,Y 37.901,Z 1002.813,A -85,B 0,C 180,E1 1427.648,E2 1427.648} C_VEL
LIN {X 0,Y 20.281,Z 1003.098,A -85,B 0,C 180,E1 1397.813,E2 1397.813} C_VEL
LIN {X 0,Y 16.146,Z 1002.507,A -85,B 0,C 180,E1 1353.658,E2 1353.658} C_VEL
LIN {X 0,Y 16.764,Z 1001.796,A -85,B 0,C 180,E1 1325.438,E2 1325.438} C_VEL
LIN {X 0,Y 26.582,Z 999.475,A -85,B 0,C 180,E1 1285.638,E2 1285.638} C_VEL
LIN {X 0,Y 45.319,Z 995.252,A -85,B 0,C 180,E1 1267.204,E2 1267.204} C_VEL
LIN {X 0,Y 65.963,Z 989.212,A -85,B 0,C 180,E1 1259.279,E2 1259.279} C_VEL
LIN {X 0,Y 87.301,Z 981.564,A -85,B 0,C 180,E1 1254.891,E2 1254.891} C_VEL
LIN {X 0,Y 107.948,Z 972.422,A -85,B 0,C 180,E1 1252.203,E2 1252.203} C_VEL
LIN {X 0,Y 129.833,Z 960.867,A -85,B 0,C 180,E1 1250.22,E2 1250.22} C_VEL
LIN {X 0,Y 148.699,Z 949.167,A -85,B 0,C 180,E1 1248.952,E2 1248.952} C_VEL
LIN {X 0,Y 167.636,Z 935.494,A -85,B 0,C 180,E1 1247.945,E2 1247.945} C_VEL
LIN {X 0,Y 186.094,Z 920.22,A -85,B 0,C 180,E1 1247.154,E2 1247.154} C_VEL
LIN {X 0,Y 202.999,Z 903.903,A -85,B 0,C 180,E1 1246.553,E2 1246.553} C_VEL
LIN {X 0,Y 217.424,Z 888.211,A -85,B 0,C 180,E1 1246.121,E2 1246.121} C_VEL
LIN {X 0,Y 220.931,Z 889.501,A -85,B 0,C 180,E1 1246.021,E2 1246.021} C_VEL
LIN {X 0,Y 220.931,Z 947.038,A -85,B 0,C 180,E1 1246.021,E2 1246.021} C_VEL
LIN {X 0,Y 170.712,Z 947.038,A -85,B 0,C 180,E1 1245.736,E2 1245.736} C_VEL
LIN {X 0,Y 168.713,Z 945.038,A -85,B 0,C 180,E1 1245.721,E2 1245.721} C_VEL
LIN {X 0,Y 168.713,Z 938.183,A -85,B 0,C 180,E1 1245.721,E2 1245.721} C_VEL
LIN {X 0,Y 165.906,Z 936.531,A -85,B 0,C 180,E1 1245.249,E2 1245.249} C_VEL
LIN {X 0,Y 146.322,Z 950.217,A -85,B 0,C 180,E1 1244.418,E2 1244.418} C_VEL
LIN {X 0,Y 126.223,Z 962.314,A -85,B 0,C 180,E1 1243.377,E2 1243.377} C_VEL
LIN {X 0,Y 105.114,Z 972.906,A -85,B 0,C 180,E1 1241.968,E2 1241.968} C_VEL
LIN {X 0,Y 83.011,Z 982.173,A -85,B 0,C 180,E1 1239.9,E2 1239.9} C_VEL
LIN {X 0,Y 62.933,Z 988.955,A -85,B 0,C 180,E1 1237.068,E2 1237.068} C_VEL
LIN {X 0,Y 39.949,Z 995.057,A -85,B 0,C 180,E1 1231.068,E2 1231.068} C_VEL
LIN {X 0,Y 21.424,Z 998.735,A -85,B 0,C 180,E1 1218.182,E2 1218.182} C_VEL
LIN {X 0,Y 8.897,Z 1000.971,A -85,B 0,C 180,E1 1169.804,E2 1169.804} C_VEL
LIN {X 0,Y 8.769,Z 1001.719,A -85,B 0,C 180,E1 1116.72,E2 1116.72} C_VEL
LIN {X 0,Y 20.337,Z 1002.766,A -85,B 0,C 180,E1 1067.779,E2 1067.779} C_VEL
LIN {X 0,Y 8.185,Z 1002.122,A -85,B 0,C 180,E1 1002.376,E2 1002.376} C_VEL
LIN {X 0,Y 8.361,Z 1001.743,A -85,B 0,C 180,E1 969.199,E2 969.199} C_VEL
LIN {X 0,Y 21.42,Z 999.364,A -85,B 0,C 180,E1 910.75,E2 910.75} C_VEL
LIN {X 0,Y 39.98,Z 995.656,A -85,B 0,C 180,E1 898.309,E2 898.309} C_VEL
LIN {X 0,Y 62.648,Z 989.561,A -85,B 0,C 180,E1 892.661,E2 892.661} C_VEL
LIN {X 0,Y 84.276,Z 982.146,A -85,B 0,C 180,E1 889.84,E2 889.84} C_VEL
LIN {X 0,Y 106.058,Z 972.781,A -85,B 0,C 180,E1 888.027,E2 888.027} C_VEL
LIN {X 0,Y 127.322,Z 961.882,A -85,B 0,C 180,E1 886.778,E2 886.778} C_VEL
LIN {X 0,Y 146.33,Z 950.324,A -85,B 0,C 180,E1 885.936,E2 885.936} C_VEL
LIN {X 0,Y 165.906,Z 936.531,A -85,B 0,C 180,E1 885.249,E2 885.249} C_VEL
LIN {X 0,Y 169.115,Z 938.111,A -85,B 0,C 180,E1 885.138,E2 885.138} C_VEL
LIN {X 0,Y 169.115,Z 996.325,A -85,B 0,C 180,E1 885.138,E2 885.138} C_VEL
LIN {X 0,Y 75.431,Z 996.325,A -85,B 0,C 180,E1 885.578,E2 885.578} C_VEL
LIN {X 0,Y 73.432,Z 994.325,A -85,B 0,C 180,E1 885.599,E2 885.599} C_VEL
LIN {X 0,Y 73.432,Z 988.486,A -85,B 0,C 180,E1 885.599,E2 885.599} C_VEL
LIN {X 0,Y 71.033,Z 986.565,A -85,B 0,C 180,E1 884.897,E2 884.897} C_VEL
LIN {X 0,Y 48.989,Z 992.908,A -85,B 0,C 180,E1 883.458,E2 883.458} C_VEL
LIN {X 0,Y 26.377,Z 997.851,A -85,B 0,C 180,E1 881.169,E2 881.169} C_VEL
LIN {X 0,Y 7.585,Z 1000.642,A -85,B 0,C 180,E1 876.729,E2 876.729} C_VEL
LIN {X 0,Y 0.305,Z 1001.586,A -85,B 0,C 180,E1 1054.081,E2 1054.081} C_VEL
LIN {X 0,Y 15.218,Z 999.763,A -85,B 0,C 180,E1 889.576,E2 889.576} C_VEL
LIN {X 0,Y 35.881,Z 996.044,A -85,B 0,C 180,E1 887.017,E2 887.017} C_VEL
LIN {X 0,Y 57.789,Z 990.659,A -85,B 0,C 180,E1 885.544,E2 885.544} C_VEL
LIN {X 0,Y 71.033,Z 986.565,A -85,B 0,C 180,E1 884.897,E2 884.897} C_VEL
LIN {X 0,Y 73.645,Z 988.468,A -85,B 0,C 180,E1 884.793,E2 884.793} C_VEL
LIN {X 0,Y 73.645,Z 1028,A -85,B 0,C 180,E1 884.793,E2 884.793} C_VEL
LIN {X 0,Y 73.645,Z 1028,A -85,B 0,C 180,E1 884.793,E2 884.793}

QRS_NEXT_CUT()

QRS_NEXT()
QRS_HOME()

END
